// TwinCAT 3 PLC project FsControllerToolbox
// Title: FsControllerToolbox
// Company: FisoThemes
// Author: Goodwill Mzumala
// ProjectVersion: 0.4.0
// Description: A library of composable building blocks for modelling and building control systems in TwinCAT.
// ProgramVersion: 3.1.4024.0
// libraries:
//   FsCommon, * (FisoThemes)
//   Tc2_Math, * (Beckhoff Automation GmbH)
//   Tc2_Standard, * (Beckhoff Automation GmbH)
//   Tc2_System, * (Beckhoff Automation GmbH)
//   Tc3_Module, * (Beckhoff Automation GmbH)
// project tree:
//   Conditioning/DUTs/ E_DeadbandMode.TcTLEO
//   Conditioning/ FB_Clamp.TcPOU, FB_Deadband.TcPOU, FB_Hysteresis.TcPOU, FB_RateLimiter.TcPOU
//   Control/DUTs/ E_AntiWindupMode.TcTLEO, E_ControllerMode.TcTLEO
//   Control/ FB_ClampingIntegrator.TcPOU, FB_Differentiator.TcPOU, FB_ExtendedStateObserver.TcPOU (not stored), FB_Integrator.TcPOU, FB_LADRC.TcPOU (not stored), FB_LinearStateErrorFeedback.TcPOU, FB_PID.TcPOU (not stored), FB_ProportionalGain.TcPOU, FB_TrackingIntegrator.TcPOU
//   Filter/ FB_FirstOrderIIRFilter.TcPOU
//   / PlcTask.TcTTO
//   Internal/ PLAYGROUND.TcPOU (not stored)
//   Project Information/ F_GetCompany.TcPOU, F_GetTitle.TcPOU, F_GetVersion.TcPOU
//   Shared/ FB_SiComponent.TcPOU, FB_SisoComponent.TcPOU, FB_SoComponent.TcPOU
//   Shared/ITFs/ I_Bounded.TcIO, I_Component.TcIO, I_Resettable.TcIO, I_SiComponent.TcIO, I_SisoComponent.TcIO, I_SoComponent.TcIO
//   Signals/DUTs/ E_RampDirection.TcTLEO
//   Signals/ FB_GaussianNoise.TcPOU, FB_PeriodicSignal.TcPOU, FB_PWM.TcPOU, FB_Ramp.TcPOU, FB_RampProfile.TcPOU, FB_SawtoothWave.TcPOU, FB_SineWave.TcPOU, FB_SquareWave.TcPOU, FB_TriangleWave.TcPOU, FB_WhiteNoise.TcPOU
//   Signals/ITFs/ I_PeriodicSignal.TcIO
//   Simulation/ FB_FirstOrderPlant.TcPOU, FB_PadeDelay.TcPOU, FB_SecondOrderPlant.TcPOU
//   Transform/ FB_Bias.TcPOU, FB_Gain.TcPOU, FB_LinearScaler.TcPOU, FB_Quantizer.TcPOU
//   Version/ Global_Version.TcGVL
// real-time tasks:
//   TASK PlcTask: cycle T#10ms, priority 20, ADS port 350
//   TASK PlcTestTask: cycle T#10ms, priority 21, ADS port 351

CONFIGURATION FsControllerToolbox
    RESOURCE PLC ON TwinCAT3
        TASK PlcTask(INTERVAL := T#10ms, PRIORITY := 20);
        PROGRAM PLAYGROUND WITH PlcTask : PLAYGROUND;
    END_RESOURCE
END_CONFIGURATION

// ---- Conditioning/DUTs/E_DeadbandMode.TcTLEO
(*
Specifies the behaviour of :itf:`FB_Deadband` when the input is within the band.
*)
{attribute 'qualified_only'}
{attribute 'strict'}
{attribute 'to_string'}
TYPE E_DeadbandMode :
(
	Hold := 0, // Output holds its last value while the input is within the band.
	Zero := 1  // Output is set to zero while the input is within the band.
)BYTE;
END_TYPE

// ---- Control/DUTs/E_AntiWindupMode.TcTLEO
(*
Specifies the anti-windup behaviour of :class:`FB_ClampingIntegrator` when
saturation is detected via :attr:`~FB_ClampingIntegrator.ComparitorInput`.
*)
{attribute 'qualified_only'}
{attribute 'strict'}
{attribute 'to_string'}
TYPE E_AntiWindupMode :
(
	// Holds the integrator output at its current value while saturation is active.
	Hold := 0,
	// Zeroes the integrator output on the rising edge of saturation detection.
	Off  := 1
)BYTE;
END_TYPE

// ---- Control/DUTs/E_ControllerMode.TcTLEO
(* Specifies the operating mode of a controller. *)
{attribute 'qualified_only'}
{attribute 'strict'}
{attribute 'to_string'}
TYPE E_ControllerMode :
(
	// Output is computed from Setpoint and Feedback using the controller's algorithm.
	Auto 	:= 0,
	// Output tracks Setpoint directly.
	Manual	:= 1
)BYTE;
END_TYPE

// ---- Signals/DUTs/E_RampDirection.TcTLEO
(* Specifies the direction of a ramping signal. *)
{attribute 'qualified_only'}
{attribute 'strict'}
{attribute 'to_string'}
TYPE E_RampDirection :
(
	Rising   := 0, // Output increases over time.
	Falling  := 1  // Output decreases over time.
)BYTE;
END_TYPE

// ---- Version/Global_Version.TcGVL
{attribute 'TcGenerated'}
{attribute 'no-analysis'}
{attribute 'linkalways'}
// This function has been automatically generated from the project information.
VAR_GLOBAL CONSTANT
	{attribute 'const_non_replaced'}
	stLibVersion_FsControllerToolbox : ST_LibVersion := (iMajor := 0, iMinor := 4, iBuild := 0, iRevision := 0, nFlags := 0, sVersion := '0.4.0');
END_VAR

// ---- Shared/ITFs/I_Bounded.TcIO
(*
Exposes configurable upper and lower bounds for blocks with clamped output.

Implemented by blocks such as :class:`FB_ClampingIntegrator` and :class:`FB_Clamp`
to allow external configuration of their output limits.
*)
INTERFACE I_Bounded EXTENDS I_Component

(*
Gets or sets the upper bound.

This value could be clamped to be greater than or equal to :attr:`Minimum`.
Thus it is best practice to set this before :attr:`Minimum` to ensure the 
guard applies correctly.
*)
PROPERTY Maximum : LREAL
GET
END_GET
SET
END_SET
END_PROPERTY

(*
Gets or sets the lower bound.

This value could be clamped to be less than or equal to :attr:`Maximum`.
Thus it is best practice to set :attr:`Maximum` before this property to 
ensure the guard applies correctly.
*)
PROPERTY Minimum : LREAL
GET
END_GET
SET
END_SET
END_PROPERTY

END_INTERFACE

// ---- Shared/ITFs/I_Component.TcIO
(*
Base interface for all FsControllerToolbox components.

Extends ``__SYSTEM.IQueryInterface`` to allow runtime type checking via
``__QUERYINTERFACE``.
*)
INTERFACE I_Component EXTENDS __SYSTEM.IQueryInterface

END_INTERFACE

// ---- Shared/ITFs/I_Resettable.TcIO
(*
Interface for components that can be returned to a known initial state.

Implementors must define :meth:`Reset` to clear any internal state, such as
accumulators, filter history, or elapsed time, and restore the output to its
initial condition.
*)
INTERFACE I_Resettable EXTENDS __SYSTEM.IQueryInterface

(* Clears internal state and restores the component to its initial condition. *)
METHOD Reset
VAR_INPUT
END_VAR
END_METHOD

END_INTERFACE

// ---- Shared/ITFs/I_SiComponent.TcIO
(*
Interface for single-input controller toolbox components.

Implementors expose a write-only :attr:`Input` property. For components that
also produce an output signal, use :itf:`I_SisoComponent` instead.
*)
INTERFACE I_SiComponent

// Gets or sets the input to the component.
PROPERTY Input : LREAL
GET
END_GET
SET
END_SET
END_PROPERTY

END_INTERFACE

// ---- Shared/ITFs/I_SisoComponent.TcIO
(*
Interface for single-input single-output controller toolbox components.

Implementors expose a writable :attr:`Input` and a read-only :attr:`Output`,
both as ``LREAL``.
*)
INTERFACE I_SisoComponent EXTENDS I_Component

// Gets or sets the input to the component.
PROPERTY Input : LREAL
GET
END_GET
SET
END_SET
END_PROPERTY

// Gets the output produced by the component.
PROPERTY Output : LREAL
GET
END_GET
END_PROPERTY

END_INTERFACE

// ---- Shared/ITFs/I_SoComponent.TcIO
(*
Interface for single-output controller toolbox components.

Implementors expose a read-only :attr:`Output` property. For components that
also accept an input signal, use :itf:`I_SisoComponent` instead.
*)
INTERFACE I_SoComponent EXTENDS I_Component

// Gets the output produced by the component.
PROPERTY Output : LREAL
GET
END_GET
END_PROPERTY

END_INTERFACE

// ---- Signals/ITFs/I_PeriodicSignal.TcIO
(*
Base interface for periodic signal generators.

Implementors produce a cyclic output defined by :attr:`Period`, :attr:`Amplitude`,
:attr:`Bias`, and :attr:`Phase`.
*)
INTERFACE I_PeriodicSignal EXTENDS I_SoComponent

(*
Gets or sets the amplitude. 

The output swings between ``Bias + Amplitude`` and ``Bias - Amplitude``.
*)
PROPERTY Amplitude : LREAL
GET
END_GET
SET
END_SET
END_PROPERTY

(*
Gets or sets the bias.

This is a fixed offset added to the output, shifting the wave up or down.
*)
PROPERTY Bias : LREAL
GET
END_GET
SET
END_SET
END_PROPERTY

(* 
Gets or sets the period. 

This is the time taken to complete one full cycle.
*)
PROPERTY Period : LTIME
GET
END_GET
SET
END_SET
END_PROPERTY

(*
Gets or sets the phase offset in radians.

This shifts the wave horizontally. Negative values shift in the opposite direction.
*)
PROPERTY Phase : LREAL
GET
END_GET
SET
END_SET
END_PROPERTY

END_INTERFACE

// ---- Conditioning/FB_Clamp.TcPOU
(*
Clamps the input signal to the range [:attr:`Minimum`, :attr:`Maximum`].

Any input below :attr:`Minimum` is set to :attr:`Minimum`. Any input above
:attr:`Maximum` is set to :attr:`Maximum`. Inputs within the range pass
through unchanged.

.. note::
   The block is ``FINAL`` and must be instantiated, not extended.
   Use ``FB_init`` to set :attr:`fMaximum` and :attr:`fMinimum` at declaration time.
*)
{attribute 'enable_dynamic_creation'}
{attribute 'no_explicit_call' := 'direct call for this function block is not allowed'}
FUNCTION_BLOCK FINAL FB_Clamp EXTENDS FB_SisoComponent
IMPLEMENTS FsCommon.I_Runnable, I_Bounded
VAR
	_fMaximum  : LREAL; // Upper clamp bound. Clamped to >= Minimum.
	_fMinimum  : LREAL; // Lower clamp bound. Clamped to <= Maximum.
	_fResidual : LREAL; // Difference between the unclamped input and the clamped output.
END_VAR

METHOD FB_init : BOOL
VAR_INPUT
	bInitRetains : BOOL; // if TRUE, the retain variables are initialized (warm start / cold start)
	bInCopyCode  : BOOL;  // if TRUE, the instance afterwards gets moved into the copy code (online change)
	fMaximum     : LREAL; // Upper clamp bound.
	fMinimum     : LREAL; // Lower clamp bound.
END_VAR
THIS^.Maximum := fMaximum;
THIS^.Minimum := fMinimum;
END_METHOD

(*
Gets or sets the upper clamp bound.

Internally clamped to be greater than or equal to :attr:`Minimum`.
Set this before :attr:`Minimum` to ensure the guard applies correctly.
*)
PROPERTY Maximum : LREAL
GET
Maximum := THIS^._fMaximum;
END_GET
SET
THIS^._fMaximum := MAX(THIS^._fMinimum, Maximum);
END_SET
END_PROPERTY

(*
Gets or sets the lower clamp bound.

Internally clamped to be less than or equal to :attr:`Maximum`.
Set :attr:`Maximum` before this property to ensure the guard applies correctly.
*)
PROPERTY Minimum : LREAL
GET
Minimum := THIS^._fMinimum;
END_GET
SET
THIS^._fMinimum := MIN(THIS^._fMaximum, Minimum);
END_SET
END_PROPERTY

(* Gets the difference between the unclamped input and the clamped output. Zero when the input is within [:attr:`Minimum`, :attr:`Maximum`]. *)
PROPERTY Residual : LREAL
GET
Residual := THIS^._fResidual;
END_GET
END_PROPERTY

(* Clamps the current input to [:attr:`Minimum`, :attr:`Maximum`]. *)
METHOD Run
VAR_INPUT
END_VAR
THIS^._fOutput 	 := LIMIT(THIS^._fMinimum, THIS^._fInput, THIS^._fMaximum);
THIS^._fResidual := THIS^._fInput - THIS^._fOutput;
END_METHOD

END_FUNCTION_BLOCK

// ---- Shared/FB_SisoComponent.TcPOU
(*
Abstract function block providing :attr:`Input` and :attr:`Output` properties
for single-input single-output controller toolbox components.

.. NOTE::
   Direct calls to this function block are not permitted (``no_explicit_call``).
*)
{attribute 'no_explicit_call' := 'direct call for this function block is not allowed'}
FUNCTION_BLOCK ABSTRACT FB_SisoComponent
IMPLEMENTS I_SisoComponent, I_SiComponent, I_SoComponent
VAR
	_fInput 	: LREAL;
	_fOutput 	: LREAL;
END_VAR

(* Gets or sets the input to the component.*)
PROPERTY Input : LREAL
GET
Input := THIS^._fInput;
END_GET
SET
THIS^._fInput := Input;
END_SET
END_PROPERTY

(* Gets the output produced by the component.*)
PROPERTY Output : LREAL
GET
Output := THIS^._fOutput;
END_GET
END_PROPERTY

END_FUNCTION_BLOCK

// ---- Conditioning/FB_Deadband.TcPOU
(*
Suppresses small input signals within a configurable band.

When the input falls within [:attr:`Minimum`, :attr:`Maximum`], the output
is either zeroed or held at its last value depending on :attr:`Mode`. Outside
the band the input passes through unchanged.

.. note::
   The block is ``FINAL`` and must be instantiated, not extended.
   Use ``FB_init`` to set :attr:`fMinimum`, :attr:`fMaximum`, and :attr:`eMode`
   at declaration time.
*)
{attribute 'enable_dynamic_creation'}
{attribute 'no_explicit_call' := 'direct call for this function block is not allowed'}
FUNCTION_BLOCK FINAL FB_Deadband EXTENDS FB_SisoComponent
IMPLEMENTS FsCommon.I_Runnable, I_Resettable
VAR
	_fMinimum  : LREAL; // Lower bound of the deadband. Clamped to <= Maximum.
	_fMaximum  : LREAL; // Upper bound of the deadband. Clamped to >= Minimum.
	_eMode     : E_DeadbandMode; // Output behaviour when input is within the band.
	_bIsActive : BOOL; // TRUE when input is within deadband [Minimum..:=Maximum].
END_VAR

METHOD FB_init : BOOL
VAR_INPUT
	bInitRetains : BOOL;  // if TRUE, the retain variables are initialized (warm start / cold start)
	bInCopyCode  : BOOL;  // if TRUE, the instance afterwards gets moved into the copy code (online change)
	fMaximum     : LREAL; // Upper bound of the deadband.
	fMinimum     : LREAL; // Lower bound of the deadband.
	eMode        : E_DeadbandMode; // Output behaviour when the input is within the band.
END_VAR
THIS^.Maximum  := fMaximum;
THIS^.Minimum  := fMinimum;
THIS^._eMode   := eMode;
END_METHOD

(*
Gets whether the input is within the deadband's bounds.

``TRUE`` when the output is being held or zeroed.
*)
PROPERTY IsActive : BOOL
GET
IsActive := THIS^._bIsActive;
END_GET
END_PROPERTY

(*
Gets or sets the upper bound of the deadband.

Internally clamped to be greater than or equal to :attr:`Minimum`.
Set this before :attr:`Minimum` to ensure the guard applies correctly.
*)
PROPERTY Maximum : LREAL
GET
Maximum := THIS^._fMaximum;
END_GET
SET
THIS^._fMaximum := MAX(THIS^._fMinimum, Maximum);
END_SET
END_PROPERTY

(*
Gets or sets the lower bound of the deadband.

Internally clamped to be less than or equal to :attr:`Maximum`.
Set :attr:`Maximum` before this property to ensure the guard applies correctly.
*)
PROPERTY Minimum : LREAL
GET
Minimum := THIS^._fMinimum;
END_GET
SET
THIS^._fMinimum := MIN(THIS^._fMaximum, Minimum);
END_SET
END_PROPERTY

(*
Gets or sets the output behaviour when the input is within the band.

:attr:`~E_DeadbandMode.Zero` sets the output to zero. 
:attr:`~E_DeadbandMode.Hold` retains the last output value. 

Changes take effect on th next :meth:`Run` call.
*)
PROPERTY Mode : E_DeadbandMode
GET
Mode := THIS^._eMode;
END_GET
SET
THIS^._eMode := Mode;
END_SET
END_PROPERTY

(* 
Resets the output to a value consistent with the current mode. 

In :attr:`~E_DeadbandMode.Zero` mode the output is set to zero.
In :attr:`~E_DeadbandMode.Hold` mode the output is set to the current input.
*)
METHOD Reset
VAR_INPUT
END_VAR
CASE THIS^._eMode OF
	E_DeadbandMode.Hold:
		THIS^._fOutput := THIS^._fInput;
	E_DeadbandMode.Zero:
		THIS^._fOutput := 0;
END_CASE
END_METHOD

(* Applies the deadband to the current input. *)
METHOD Run
VAR_INPUT
END_VAR
THIS^._fMaximum := MAX(THIS^._fMinimum, THIS^._fMaximum);
THIS^._fMinimum := MIN(THIS^._fMinimum, THIS^._fMaximum);

THIS^._bIsActive := THIS^._fInput >= THIS^._fMinimum AND THIS^._fInput <= THIS^._fMaximum;

IF THIS^._bIsActive  THEN
    CASE THIS^._eMode OF
        E_DeadbandMode.Zero:
            THIS^._fOutput := 0;
        E_DeadbandMode.Hold:
            ; // Output retains its last value.
    END_CASE
ELSE
    THIS^._fOutput := THIS^._fInput;
END_IF
END_METHOD

END_FUNCTION_BLOCK

// ---- Conditioning/FB_Hysteresis.TcPOU
(*
Implements a hysteresis controller with two thresholds and latching behaviour.

The output switches low when the input rises above :attr:`UpperThreshold` and
switches high when the input falls below :attr:`LowerThreshold`. Between the
two thresholds the output latches at its current state.

This convention suits heating applications, the output drives a heater that
turns on when the process falls below the lower threshold and off when it
exceeds the upper threshold.

.. note::
   The block is ``FINAL`` and must be instantiated, not extended.
   Use ``FB_init`` to set :attr:`fUpperThreshold` and :attr:`fLowerThreshold`
   at declaration time.
*)
{attribute 'no_assign'}
{attribute 'enable_dynamic_creation'}
{attribute 'no_explicit_call' := 'direct call for this function block is not allowed'}
FUNCTION_BLOCK FINAL FB_Hysteresis EXTENDS FB_SiComponent
IMPLEMENTS FsCommon.I_Runnable, I_Resettable
VAR
	_fUpperThreshold : LREAL; // Input level above which the output switches low.
	_fLowerThreshold : LREAL; // Input level below which the output switches high.
	_bOutput         : BOOL;  // Current output state.
END_VAR

METHOD FB_init : BOOL
VAR_INPUT
	bInitRetains 	 : BOOL; // if TRUE, the retain variables are initialized (warm start / cold start)
	bInCopyCode 	 : BOOL;  // if TRUE, the instance afterwards gets moved into the copy code (online change)
	fUpperThreshold  : LREAL; // Input level above which the output switches low.
	fLowerThreshold  : LREAL; // Input level below which the output switches high.
END_VAR
THIS^._fUpperThreshold := fUpperThreshold;
THIS^._fLowerThreshold := fLowerThreshold;
END_METHOD

(*
Gets or sets the lower threshold.

When the input falls below this value the output switches high. Must be less
than :attr:`UpperThreshold` for correct operation.
*)
PROPERTY LowerThreshold : LREAL
GET
LowerThreshold := THIS^._fLowerThreshold;
END_GET
SET
THIS^._fLowerThreshold := LowerThreshold;
END_SET
END_PROPERTY

(*
Gets the current output state. 

TRUE when the process is below :attr:`LowerThreshold`.
FALSE when above :attr:`UpperThreshold`.
*)
PROPERTY Output : BOOL
GET
Output := THIS^._bOutput;
END_GET
END_PROPERTY

(*
Evaluates the current input against the thresholds and sets the output immediately,
rather than waiting for the input to cross a threshold.

If the input is above :attr:`UpperThreshold` the output is set low. If below
:attr:`LowerThreshold` the output is set high. If between the two thresholds
the output defaults to low as a safe state.
*)
METHOD Reset
VAR_INPUT
END_VAR
THIS^._bOutput := THIS^._fInput < THIS^._fLowerThreshold;
END_METHOD

(* Evaluates the input against the thresholds and updates the output. *)
METHOD Run
VAR_INPUT
END_VAR
IF THIS^._fInput > THIS^._fUpperThreshold THEN
	THIS^._bOutput := FALSE;
ELSIF THIS^._fInput < THIS^._fLowerThreshold THEN
	THIS^._bOutput := TRUE;
END_IF
END_METHOD

(*
Gets or sets the upper threshold.

When the input rises above this value the output switches low. Must be greater
than :attr:`LowerThreshold` for correct operation.
*)
PROPERTY UpperThreshold : LREAL
GET
UpperThreshold := THIS^._fUpperThreshold;
END_GET
SET
THIS^._fUpperThreshold := UpperThreshold;
END_SET
END_PROPERTY

END_FUNCTION_BLOCK

// ---- Shared/FB_SiComponent.TcPOU
(*
Abstract function block providing an :attr:`Input` property for single-input
controller toolbox components.

Concrete implementations read from ``_fInput`` to consume the signal written
by the caller.

.. note::
   Direct calls to this function block are not permitted (``no_explicit_call``).
   Extend it and call the derived block instead.
*)
{attribute 'no_explicit_call' := 'direct call for this function block is not allowed'}
FUNCTION_BLOCK ABSTRACT FB_SiComponent
IMPLEMENTS I_SiComponent
VAR
    _fInput : LREAL;
END_VAR

(* Gets or sets the input to the component.*)
PROPERTY Input : LREAL
GET
Input := THIS^._fInput;
END_GET
SET
THIS^._fInput := Input;
END_SET
END_PROPERTY

END_FUNCTION_BLOCK

// ---- Conditioning/FB_RateLimiter.TcPOU
(*
Limits the rate of change of the input signal.

The output tracks the input but cannot change faster than :attr:`RisingLimit`
units per second when increasing, or :attr:`FallingLimit` units per second when
decreasing. A limit of zero removes the restriction in that direction, allowing
the output to change freely.

Calling :meth:`Reset` snaps the output to the current input immediately.

.. note::
   The block is ``FINAL`` and must be instantiated, not extended.
   Use ``FB_init`` to set :attr:`fRisingLimit` and :attr:`fFallingLimit` at
   declaration time.
*)
{attribute 'enable_dynamic_creation'}
{attribute 'no_explicit_call' := 'direct call for this function block is not allowed'}
FUNCTION_BLOCK FINAL FB_RateLimiter EXTENDS FB_SisoComponent
IMPLEMENTS FsCommon.I_Runnable, I_Resettable
VAR
	_fRisingLimit  : LREAL; // Maximum rate of increase in units per second. Zero means no limit.
	_fFallingLimit : LREAL; // Maximum rate of decrease in units per second. Zero means no limit.
END_VAR

(*
Gets or sets the maximum rate of decrease in units per second.

The output will not fall faster than this value regardless of how quickly
the input changes. A value of zero removes the falling limit entirely.
Values below zero are clamped to zero.
*)
PROPERTY FallingLimit : LREAL
GET
FallingLimit := THIS^._fFallingLimit;
END_GET
SET
THIS^._fFallingLimit := MAX(0, FallingLimit);
END_SET
END_PROPERTY

METHOD FB_init : BOOL
VAR_INPUT
	bInitRetains   : BOOL; // if TRUE, the retain variables are initialized (warm start / cold start)
	bInCopyCode    : BOOL;  // if TRUE, the instance afterwards gets moved into the copy code (online change)
	fRisingLimit   : LREAL; // Maximum rate of increase in units per second. Zero means no limit.
	fFallingLimit  : LREAL; // Maximum rate of decrease in units per second. Zero means no limit.
END_VAR
THIS^.RisingLimit  := fRisingLimit;
THIS^.FallingLimit := fFallingLimit;
END_METHOD

(* Snaps the output to the current input, bypassing the rate limit. *)
METHOD Reset
VAR_INPUT
END_VAR
THIS^._fOutput := THIS^._fInput;
END_METHOD

(*
Gets or sets the maximum rate of increase in units per second.

The output will not rise faster than this value regardless of how quickly
the input changes. A value of zero removes the rising limit entirely.
Values below zero are clamped to zero.
*)
PROPERTY RisingLimit : LREAL
GET
RisingLimit := THIS^._fRisingLimit;
END_GET
SET
THIS^._fRisingLimit := MAX(0, RisingLimit);
END_SET
END_PROPERTY

(*
Advances the rate limiter by one time step.

.. note::
   Must be called once per cycle on a single PLC task. If the measured cycle
   time is zero the method returns early without updating the output.
*)
METHOD Run
VAR_INST
	{attribute 'hide'}
	bInit       : BOOL := TRUE;
	{attribute 'hide'}
	fT          : LREAL;
	{attribute 'hide'}
	fbTaskCycle : FsCommon.FB_PlcTaskCycleChangeDetector(0);
END_VAR
VAR
	fDelta    	: LREAL;
	fMaxDelta 	: LREAL;
END_VAR
IF bInit THEN
	fT := TO_LREAL(FsCommon.F_GetCurrentTaskCycleTime()) / TO_LREAL(LTIME#1S);
	RETURN(bInit := fT <= 0);
	fbTaskCycle.TaskIndex := FsCommon.F_GetCurrentTaskIndex();
	THIS^._fOutput := THIS^._fInput;
	RETURN;
END_IF

RETURN(NOT fbTaskCycle.HasChanged);

THIS^._fRisingLimit  := MAX(0, THIS^._fRisingLimit);
THIS^._fFallingLimit := MAX(0, THIS^._fFallingLimit);

fDelta := THIS^._fInput - THIS^._fOutput;

IF fDelta > 0 AND THIS^._fRisingLimit > 0 THEN
	fMaxDelta      := THIS^._fRisingLimit * fT;
	THIS^._fOutput := THIS^._fOutput + MIN(fDelta, fMaxDelta);
ELSIF fDelta < 0 AND THIS^._fFallingLimit > 0 THEN
	fMaxDelta      := THIS^._fFallingLimit * fT;
	THIS^._fOutput := THIS^._fOutput - MIN(ABS(fDelta), fMaxDelta);
ELSE
	THIS^._fOutput := THIS^._fInput;
END_IF
END_METHOD

END_FUNCTION_BLOCK

// ---- Control/FB_ClampingIntegrator.TcPOU
(*
Integrates the input error signal with comparator-based anti-windup.

Extends :class:`FB_Integrator` by suppressing integration when the
:attr:`ComparatorInput` indicates saturation and the input would push
further into saturation. The suppression behaviour is controlled by :attr:`Mode`.

:attr:`ComparatorInput` is typically the :attr:`~FB_Clamp.Residual` of an
:class:`FB_Clamp` block placed after the PID summation.

.. note::
   Set :attr:`Maximum` before :attr:`Minimum` to ensure the clamp guard applies
   correctly.

   Use ``FB_init`` to set :attr:`tTn` and :attr:`eMode` at declaration time.
*)
{attribute 'no_assign'}
{attribute 'enable_dynamic_creation'}
{attribute 'no_explicit_call' := 'direct call for this function block is not allowed'}
FUNCTION_BLOCK FINAL FB_ClampingIntegrator EXTENDS FB_Integrator
VAR
	_fComparatorInput  : LREAL;
	_bAntiWindupActive : BOOL; // TRUE when the output is saturated and integration is halted.
	_eMode			   : E_AntiWindupMode; // The integrator behaviour during saturation.
END_VAR

(* Gets whether the output is currently saturated and integration is halted. *)
PROPERTY AntiWindupActive : BOOL
GET
AntiWindupActive := THIS^._bAntiWindupActive;
END_GET
END_PROPERTY

(*
Gets or sets the comparator input.

This is typically the :attr:`~FB_Clamp.Residual` of an :class:`FB_Clamp` block
placed after the PID summation. A positive value indicates the unsaturated sum
exceeded the clamp maximum; a negative value indicates it fell below the clamp
minimum. When this value and :attr:`Input` have the same sign, integration is
suppressed according to :attr:`Mode`.
*)
PROPERTY ComparatorInput : LREAL
GET
ComparatorInput := THIS^._fComparatorInput;
END_GET
SET
THIS^._fComparatorInput := ComparatorInput;
END_SET
END_PROPERTY

METHOD FB_init : BOOL
VAR_INPUT
	bInitRetains : BOOL;  // if TRUE, the retain variables are initialized (warm start / cold start)
	bInCopyCode  : BOOL;  // if TRUE, the instance afterwards gets moved into the copy code (online change)
	tTn          : LTIME; // Integral action time. LTIME#0 disables integration.
	eMode		 : E_AntiWindupMode; // The integrator behaviour during saturation.
END_VAR
THIS^._eMode := eMode;
END_METHOD

(*
Gets or sets the anti-windup mode.

Controls the integrator behaviour when saturation is detected via
:attr:`ComparatorInput`. See :class:`E_AntiWindupMode` for available modes.
*)
PROPERTY Mode : E_AntiWindupMode
GET
Mode := THIS^._eMode;
END_GET
SET
THIS^._eMode := Mode;
END_SET
END_PROPERTY

(* Clears the integrator state, output, and anti-windup flag. *)
METHOD Reset
VAR_INPUT
END_VAR
THIS^._fOutput           := 0;
THIS^._bAntiWindupActive := FALSE;
END_METHOD

(*
Advances the clamping integrator by one time step.

.. note::
   Must be called once per cycle on a single PLC task. If :attr:`Tn` is
   ``LTIME#0`` the output is set to zero and anti-windup is cleared.
*)
METHOD Run
VAR_INST
	{attribute 'hide'}
	bInit       : BOOL := TRUE;
	{attribute 'hide'}
	fT          : LREAL;
	{attribute 'hide'}
	fbTaskCycle : FsCommon.FB_PlcTaskCycleChangeDetector(0);
	{attribute 'hide'}
	fbTrig 		: F_TRIG;
END_VAR
VAR
END_VAR
IF bInit THEN
	fT := TO_LREAL(FsCommon.F_GetCurrentTaskCycleTime()) / TO_LREAL(LTIME#1S);
	RETURN(bInit := fT <= 0);
	fbTaskCycle.TaskIndex := FsCommon.F_GetCurrentTaskIndex();
END_IF

RETURN(NOT fbTaskCycle.HasChanged);

THIS^._fMaximum := MAX(THIS^._fMinimum, THIS^._fMaximum);
THIS^._fMinimum := MIN(THIS^._fMinimum, THIS^._fMaximum);

IF FsCommon.F_ResetOnTrue(THIS^._bSync) THEN
	THIS^._fOutput := LIMIT(THIS^._fMinimum, THIS^._fSync, THIS^._fMaximum);
END_IF

IF THIS^._tTn = LTIME#0S THEN
	THIS^._fOutput           := 0;
	THIS^._bAntiWindupActive := FALSE;
	RETURN;
END_IF

THIS^._bAntiWindupActive := (THIS^._fComparatorInput > 0.0 AND THIS^._fInput > 0.0)
							 OR 
                            (THIS^._fComparatorInput < 0.0 AND THIS^._fInput < 0.0);
							
fbTrig(CLK := THIS^._bAntiWindupActive);
IF fbTrig.Q AND THIS^._eMode = E_AntiWindupMode.Off THEN 
	THIS^._bAntiWindupActive := TRUE;
END_IF
							
IF THIS^._bAntiWindupActive THEN
	CASE THIS^._eMode OF 
		E_AntiWindupMode.Hold:;
		E_AntiWindupMode.Off:
			THIS^._fOutput := 0.0;
	END_CASE
ELSE
	THIS^._fOutput := LIMIT(
		THIS^._fMinimum, 
		THIS^._fOutput + (1.0 / (TO_LREAL(THIS^._tTn) / TO_LREAL(LTIME#1S))) * THIS^._fInput * fT,
		THIS^._fMaximum
	);
END_IF
END_METHOD

END_FUNCTION_BLOCK

// ---- Control/FB_Integrator.TcPOU
(*
Integrates the input error signal over time.

The output accumulates the input scaled by the integral gain :math:`K_i = 1 / T_n`,
and is clamped to [:attr:`Minimum`, :attr:`Maximum`] on every cycle.
Setting :attr:`Tn` to ``LTIME#0`` disables integration, setting the output to zero.

Use :meth:`Sync` to preset the integrator state for bumpless transfer when
switching from manual to automatic mode.

.. note::
   Set :attr:`Maximum` before :attr:`Minimum` to ensure the clamp guard applies
   correctly.

   Use ``FB_init`` to set :attr:`tTn` at declaration time.
*)
{attribute 'no_assign'}
{attribute 'enable_dynamic_creation'}
{attribute 'no_explicit_call' := 'direct call for this function block is not allowed'}
FUNCTION_BLOCK FB_Integrator EXTENDS FB_SisoComponent
IMPLEMENTS FsCommon.I_Runnable, I_Resettable, I_Bounded
VAR
	_tTn   		: LTIME; // Integral action time (Tn).
	_bSync 		: BOOL;  // Triggers a bumpless transfer on the next Run call.
	_fSync 		: LREAL; // Target integrator state for bumpless transfer.
	_fMaximum   : LREAL := FsCommon.GVL_TypeValueLimits.LREAL_MAX; // Upper output clamp. Clamped to >= Minimum.
	_fMinimum   : LREAL := FsCommon.GVL_TypeValueLimits.LREAL_MIN; // Lower output clamp. Clamped to <= Maximum.
END_VAR

METHOD FB_init : BOOL
VAR_INPUT
	bInitRetains : BOOL;  // if TRUE, the retain variables are initialized (warm start / cold start)
	bInCopyCode  : BOOL;  // if TRUE, the instance afterwards gets moved into the copy code (online change)
	tTn          : LTIME; // Integral action time. LTIME#0 disables integration.
END_VAR
THIS^._tTn := tTn;
END_METHOD

(*
Gets or sets the upper output clamp.

Internally clamped to be greater than or equal to :attr:`Minimum`.
Set this before :attr:`Minimum` to ensure the guard applies correctly.
*)
PROPERTY Maximum : LREAL
GET
Maximum := THIS^._fMaximum;
END_GET
SET
THIS^._fMaximum := MAX(THIS^._fMinimum, Maximum);
END_SET
END_PROPERTY

(*
Gets or sets the lower output clamp.

Internally clamped to be less than or equal to :attr:`Maximum`.
Set :attr:`Maximum` before this property to ensure the guard applies correctly.
*)
PROPERTY Minimum : LREAL
GET
Minimum := THIS^._fMinimum;
END_GET
SET
THIS^._fMinimum := MIN(THIS^._fMaximum, Minimum);
END_SET
END_PROPERTY

(* Clears the integrator state and output. *)
METHOD Reset
VAR_INPUT
END_VAR
THIS^._fOutput := 0;
END_METHOD

(*
Advances the integrator by one time step.

.. note::
   Must be called once per cycle on a single PLC task. If :attr:`Tn` is
   ``LTIME#0`` the output is set to zero.
*)
METHOD Run
VAR_INST
	{attribute 'hide'}
	bInit       : BOOL := TRUE;
	{attribute 'hide'}
	fT          : LREAL;
	{attribute 'hide'}
	fbTaskCycle : FsCommon.FB_PlcTaskCycleChangeDetector(0);
END_VAR
IF bInit THEN
	fT := TO_LREAL(FsCommon.F_GetCurrentTaskCycleTime()) / TO_LREAL(LTIME#1S);
	RETURN(bInit := fT <= 0);
	fbTaskCycle.TaskIndex := FsCommon.F_GetCurrentTaskIndex();
END_IF

RETURN(NOT fbTaskCycle.HasChanged);

THIS^._fMaximum := MAX(THIS^._fMinimum, THIS^._fMaximum);
THIS^._fMinimum := MIN(THIS^._fMinimum, THIS^._fMaximum);

IF FsCommon.F_ResetOnTrue(THIS^._bSync) THEN
	THIS^._fOutput := THIS^._fSync;
END_IF

IF THIS^._tTn = LTIME#0S THEN
	THIS^._fOutput := 0;
	RETURN;
END_IF

THIS^._fOutput := LIMIT(
	THIS^._fMinimum, 
	THIS^._fOutput + 
		(1.0 / (TO_LREAL(THIS^._tTn) / TO_LREAL(LTIME#1S))) * THIS^._fInput * fT,
	THIS^._fMaximum
);
END_METHOD

(*
Forces the integrator state to a given value on the next :meth:`Run` call.

Use this for bumpless transfer when switching from manual to automatic mode,
to prevent a sudden jump in output.
*)
METHOD Sync
VAR_INPUT
	// Target integrator state.
	fValue : LREAL; 
END_VAR
THIS^._bSync := TRUE;
THIS^._fSync := fValue;
END_METHOD

(*
Gets or sets the integral action time (Tn).

This controls how aggressively the integrator responds to sustained error.
A shorter value increases integral action. Setting it to ``LTIME#0`` disables
integration entirely, setting the output to zero.
*)
PROPERTY Tn : LTIME
GET
Tn := THIS^._tTn;
END_GET
SET
THIS^._tTn := Tn;
END_SET
END_PROPERTY

END_FUNCTION_BLOCK

// ---- Control/FB_Differentiator.TcPOU
(*
Differentiates the input signal with an optional first-order damping filter.

The transfer function is:

.. math::

   D(s) = \frac{T_v \cdot s}{T_d \cdot s + 1}

where :math:`T_v` is :attr:`Tv` and :math:`T_d` is :attr:`Td`. The filter is
discretised using the Tustin (bilinear) method.

Setting :attr:`Tv` to ``LTIME#0`` disables the derivative term entirely.
Setting :attr:`Td` to ``LTIME#0`` removes the damping filter, giving a pure
derivative. This is not recommended in practice due to noise sensitivity.

.. note::
   If derivative kick on setpoint steps is undesirable, pass the negated
   process variable as :attr:`Input` rather than the full error. The integrator
   should still receive the full error signal.

   The block is ``FINAL`` and must be instantiated, not extended.
   Use ``FB_init`` to set :attr:`tTv` and :attr:`tTd` at declaration time.
*)
{attribute 'no_assign'}
{attribute 'enable_dynamic_creation'}
{attribute 'no_explicit_call' := 'direct call for this function block is not allowed'}
FUNCTION_BLOCK FINAL FB_Differentiator EXTENDS FB_SisoComponent
IMPLEMENTS FsCommon.I_Runnable, I_Resettable
VAR
	_tTv          : LTIME; // Rate time (Tv). Determines derivative action strength.
	_tTd          : LTIME; // Damping time (Td). Filters the derivative signal to reduce noise sensitivity.
	_fPrevInput   : LREAL; // Input from the previous cycle.
	_fFilterState : LREAL; // Internal state of the damping filter.
END_VAR

METHOD FB_init : BOOL
VAR_INPUT
	bInitRetains : BOOL; // if TRUE, the retain variables are initialized (warm start / cold start)
	bInCopyCode  : BOOL;  // if TRUE, the instance afterwards gets moved into the copy code (online change)
	tTv          : LTIME; // Rate time. T#0S disables the derivative term entirely.
	tTd          : LTIME; // Damping time. LTIME#0 means no filtering (pure derivative).
END_VAR
THIS^._tTv := tTv;
THIS^._tTd := tTd;
END_METHOD

(*
Clears the filter state and output. 
Sets the previous input to the current input to avoid a spike on the next :meth:`Run` call. 
*)
METHOD Reset
VAR_INPUT
END_VAR
THIS^._fFilterState := 0;
THIS^._fPrevInput   := THIS^._fInput;
THIS^._fOutput      := 0;
END_METHOD

(*
Advances the differentiator by one time step.

On the first call the cycle time is measured, the filter state is initialised,
and the method returns early without producing an output. This prevents a spike
caused by an uninitialised previous input.

.. note::
   Must be called once per cycle on a single PLC task. If :attr:`Tv` is
   ``LTIME#0`` the output is held at zero.
*)
METHOD Run
VAR_INST
	{attribute 'hide'}
	bInit       : BOOL := TRUE;
	{attribute 'hide'}
	fT          : LREAL;
	{attribute 'hide'}
	fbTaskCycle : FsCommon.FB_PlcTaskCycleChangeDetector(0);
END_VAR
VAR
	fTv            : LREAL;
	fTd            : LREAL;
	fDen           : LREAL;
	fAlpha         : LREAL;
	fRawDerivative : LREAL;
END_VAR
IF bInit THEN
	fT := TO_LREAL(FsCommon.F_GetCurrentTaskCycleTime()) / TO_LREAL(LTIME#1S);
	RETURN(bInit := fT <= 0);
	fbTaskCycle.TaskIndex := FsCommon.F_GetCurrentTaskIndex();
	THIS^._fPrevInput     := THIS^._fInput;
	THIS^._fFilterState   := 0;
	RETURN;
END_IF

RETURN(NOT fbTaskCycle.HasChanged);

IF THIS^._tTv = LTIME#0S THEN
	THIS^._fOutput    := 0;
	THIS^._fPrevInput := THIS^._fInput;
	RETURN;
END_IF

fTv := TO_LREAL(THIS^._tTv) / TO_LREAL(LTIME#1S);
fTd := TO_LREAL(THIS^._tTd) / TO_LREAL(LTIME#1S);

fRawDerivative := fTv * (THIS^._fInput - THIS^._fPrevInput) / fT;

IF THIS^._tTd = LTIME#0S THEN
	THIS^._fOutput := fRawDerivative;
ELSE
	fDen                := fTd + fT / 2.0;
	fAlpha              := (fTd - fT / 2.0) / fDen;
	THIS^._fFilterState := fAlpha * THIS^._fFilterState + (1.0 - fAlpha) * fRawDerivative;
	THIS^._fOutput      := THIS^._fFilterState;
END_IF

THIS^._fPrevInput := THIS^._fInput;
END_METHOD

(*
Gets or sets the damping time (Td).

This filters the derivative signal to reduce sensitivity to noise. A longer
value gives more filtering but reduces derivative effectiveness. Setting it
to ``LTIME#0`` removes the filter entirely, giving a pure derivative (not
recommended in practice due to noise sensitivity).
*)
PROPERTY Td : LTIME
GET
Td := THIS^._tTd;
END_GET
SET
THIS^._tTd := Td;
END_SET
END_PROPERTY

(*
Gets or sets the rate time (Tv).

This controls how strongly the block reacts to changes in the input. A longer
value increases derivative action. Setting it to ``LTIME#0`` disables the
derivative term entirely, holding the output at zero.
*)
PROPERTY Tv : LTIME
GET
Tv := THIS^._tTv;
END_GET
SET
THIS^._tTv := Tv;
END_SET
END_PROPERTY

END_FUNCTION_BLOCK

// ---- Control/FB_LinearStateErrorFeedback.TcPOU
(*
Computes the control output for a Linear Active Disturbance Rejection Controller (LADRC).

The control law is:

.. math::

   u_0 = \omega_c \cdot (SP - z_1) + u_i

   u = \frac{u_0 - z_2}{b_0}

where :math:`u_0` is the error feedback, :math:`u_i` is the integral correction
from an external integrator, :math:`z_2` cancels the estimated disturbance from
:class:`FB_ExtendedStateObserver`, and dividing by :attr:`B0` scales the output
to the plant's input range.

If :attr:`B0` is zero the output is held at zero.

.. note::
   The block is ``FINAL`` and must be instantiated, not extended.
   Use ``FB_init`` to set :attr:`fWc` and :attr:`fB0` at declaration time.
*)
{attribute 'no_assign'}
{attribute 'enable_dynamic_creation'}
{attribute 'no_explicit_call' := 'direct call for this function block is not allowed'}
FUNCTION_BLOCK FINAL FB_LinearStateErrorFeedback EXTENDS FB_SoComponent
IMPLEMENTS FsCommon.I_Runnable, I_Resettable
VAR
	_fWc       : LREAL; // Controller bandwidth in rad/s.
	_fB0       : LREAL; // Estimated plant gain.
	_fSetpoint : LREAL; // Desired process output (SP).
	_fZ1       : LREAL; // Estimated process output from the observer.
	_fZ2       : LREAL; // Estimated total disturbance from the observer.
	_fIntegral : LREAL; // Integral correction from the external integrator.
END_VAR

(*
Gets or sets the estimated plant gain (b0).

Must be non-zero. A value of zero disables the control output entirely.
See :attr:`~FB_ADRC.B0` for guidance on how to estimate this value.
*)
PROPERTY B0 : LREAL
GET
B0 := THIS^._fB0;
END_GET
SET
THIS^._fB0 := B0;
END_SET
END_PROPERTY

METHOD FB_init : BOOL
VAR_INPUT
	bInitRetains : BOOL; // if TRUE, the retain variables are initialized (warm start / cold start)
	bInCopyCode : BOOL;  // if TRUE, the instance afterwards gets moved into the copy code (online change)
	fWc          : LREAL; // Controller bandwidth in rad/s.
	fB0          : LREAL; // Estimated plant gain.
END_VAR
THIS^._fWc := fWc;
THIS^._fB0 := fB0;
END_METHOD

(*
Gets or sets the integral correction.

Set this to the integrator output before calling :meth:`Run`. 
*)
PROPERTY Integral : LREAL
GET
Integral := THIS^._fIntegral;
END_GET
SET
THIS^._fIntegral := Integral;
END_SET
END_PROPERTY

(* Sets the output to zero. *)
METHOD Reset
VAR_INPUT
END_VAR
THIS^._fOutput := 0;
END_METHOD

(*
Computes the control output for the current cycle.

.. note::
   Must be called once per cycle on a single PLC task.
   If :attr:`b0` is zero the output is held at zero.
*)
METHOD Run
VAR
END_VAR
RETURN(THIS^._fb0 = 0);

THIS^._fOutput :=
    ((THIS^._fWc * (THIS^._fSetpoint - THIS^._fZ1)) + THIS^._fIntegral - THIS^._fZ2)
    / THIS^._fB0;
END_METHOD

(* Gets or sets the setpoint. This is the desired process output. *)
PROPERTY Setpoint : LREAL
GET
Setpoint := THIS^._fSetpoint;
END_GET
SET
THIS^._fSetpoint := Setpoint;
END_SET
END_PROPERTY

(*
Gets or sets the controller bandwidth in rad/s.

Controls how fast the closed loop responds to setpoint changes. A higher value
gives a faster response but risks overshoot and sensitivity to noise. Start with
a low value and increase until the response is satisfactory.

For a process that should settle in roughly 10 seconds, a starting value of
``Wc = 0.5`` rad/s is reasonable.
*)
PROPERTY Wc : LREAL
GET
Wc := THIS^._fWc;
END_GET
SET
THIS^._fWc := Wc;
END_SET
END_PROPERTY

(* 
Gets or sets the estimated process output from :class:`FB_ExtendedStateObserver`. 

Set this to ``Z1`` before calling :meth:`Run`.
*)
PROPERTY Z1 : LREAL
GET
Z1 := THIS^._fZ1;
END_GET
SET
THIS^._fZ1 := Z1;
END_SET
END_PROPERTY

(*
Gets or sets the estimated total disturbance from :class:`FB_ExtendedStateObserver`. 

Set this to ``Z2`` before calling :meth:`Run`.
*)
PROPERTY Z2 : LREAL
GET
Z2 := THIS^._fZ2;
END_GET
SET
THIS^._fZ2 := Z2;
END_SET
END_PROPERTY

END_FUNCTION_BLOCK

// ---- Shared/FB_SoComponent.TcPOU
(*
Abstract function block providing an :attr:`Output` property for single-output
controller toolbox components.

Concrete implementations must call this block cyclically and write their
result to ``_fOutput``.

.. note::
   Direct calls to this function block are not permitted (``no_explicit_call``).
   Extend it and call the derived block instead.
*)
{attribute 'no_explicit_call' := 'direct call for this function block is not allowed'}
FUNCTION_BLOCK ABSTRACT FB_SoComponent
IMPLEMENTS I_SoComponent
VAR
	_fOutput : LREAL;
END_VAR

(* Gets the output produced by the component.*)
PROPERTY Output : LREAL
GET
Output := THIS^._fOutput;
END_GET
END_PROPERTY

END_FUNCTION_BLOCK

// ---- Control/FB_ProportionalGain.TcPOU
(*
Applies a proportional gain to the input error signal.

The output is computed as:

.. math::

   y = K_p \cdot e

where :math:`K_p` is :attr:`Kp` and :math:`e` is the error signal set via :attr:`Input`.

.. note::
   The block is ``FINAL`` and must be instantiated, not extended.
   Use ``FB_init`` to set :attr:`fKp` at declaration time.
*)
{attribute 'no_assign'}
{attribute 'enable_dynamic_creation'}
{attribute 'no_explicit_call' := 'direct call for this function block is not allowed'}
FUNCTION_BLOCK FINAL FB_ProportionalGain EXTENDS FB_SisoComponent
IMPLEMENTS FsCommon.I_Runnable, I_Resettable
VAR
	_fKp : LREAL; // Proportional gain.
END_VAR

METHOD FB_init : BOOL
VAR_INPUT
	bInitRetains : BOOL; // if TRUE, the retain variables are initialized (warm start / cold start)
	bInCopyCode  : BOOL;  // if TRUE, the instance afterwards gets moved into the copy code (online change)
	fKp          : LREAL; // Proportional gain.
END_VAR
THIS^._fKp := fKp;
END_METHOD

(*
Gets or sets the proportional gain.

A higher value produces a stronger response to error but may cause overshoot.
A lower value produces a more gradual response. A value of 0 disables the
proportional term entirely.
*)
PROPERTY Kp : LREAL
GET
Kp := THIS^._fKp;
END_GET
SET
THIS^._fKp := Kp;
END_SET
END_PROPERTY

(* Sets the output to zero. Takes effect until the next :meth:`Run` call. *)
METHOD Reset
VAR_INPUT
END_VAR
THIS^._fOutput := 0;
END_METHOD

(*
Computes the proportional output for the current cycle.

.. note::
   Must be called once per cycle on a single PLC task.
*)
METHOD Run
VAR_INPUT
END_VAR
THIS^._fOutput := THIS^._fKp * THIS^._fInput;
END_METHOD

END_FUNCTION_BLOCK

// ---- Control/FB_TrackingIntegrator.TcPOU
(*
Integrates the input error signal with back-calculation anti-windup.

Extends :class:`FB_Integrator` by accepting an external comparator input,
typically the :attr:`~FB_Clamp.Residual` of an :class:`FB_Clamp` block, to
unwind the integrator gradually when the output is saturated. The residual is
scaled by ``1 / Tt`` and subtracted from the integrator input each cycle.

A typical wiring pattern:

.. code-block:: pascal

   fbI.Input           := fbP.Output; // Standard form. Use fError for parallel form.
   fbI.ComparatorInput := fbClamp.Residual;
   fbI.Run();
   fbClamp.Input := fbP.Output + fbI.Output + fbD.Output;
   fbClamp.Run();

.. note::
   Set :attr:`Maximum` before :attr:`Minimum` to ensure the clamp guard applies
   correctly.

   Use ``FB_init`` to set :attr:`tTn` and :attr:`tTt` at declaration time.
*)
{attribute 'no_assign'}
{attribute 'enable_dynamic_creation'}
{attribute 'no_explicit_call' := 'direct call for this function block is not allowed'}
FUNCTION_BLOCK FINAL FB_TrackingIntegrator EXTENDS FB_Integrator
VAR
	_fComparatorInput  : LREAL; // External residual signal for back-calculation anti-windup.
	_tTt 			   : LTIME; // Tracking time constant (Tt). Controls how quickly the integrator unwinds.
END_VAR

(*
Gets or sets the comparator input.

This is typically the :attr:`~FB_Clamp.Residual` of an :class:`FB_Clamp` block
placed after the PID summation, passed directly without negation. The block
subtracts the scaled residual from the integrator input internally to unwind
the integrator when the output is saturated.

A positive value indicates the unsaturated sum exceeded the clamp maximum.
A negative value indicates it fell below the clamp minimum.
*)
PROPERTY ComparatorInput : LREAL
GET
ComparatorInput := THIS^._fComparatorInput;
END_GET
SET
THIS^._fComparatorInput := ComparatorInput;
END_SET
END_PROPERTY

METHOD FB_init : BOOL
VAR_INPUT
	bInitRetains : BOOL;  // if TRUE, the retain variables are initialized (warm start / cold start)
	bInCopyCode  : BOOL;  // if TRUE, the instance afterwards gets moved into the copy code (online change)
	tTn          : LTIME; // Integral action time. LTIME#0 disables integration.
	tTt 		 : LTIME; // Tracking time constant (Tt). A typical starting value is SQRT(Tn * Td).
END_VAR
THIS^._tTt := tTt;
END_METHOD

(*
Advances the tracking integrator by one time step.

.. note::
   Must be called once per cycle on a single PLC task. If :attr:`Tn` is
   ``LTIME#0`` the output is set to zero. If :attr:`Tt` is ``LTIME#0``
   the back-calculation correction is disabled.
*)
METHOD Run
VAR_INST
	{attribute 'hide'}
	bInit       : BOOL := TRUE;
	{attribute 'hide'}
	fT          : LREAL;
	{attribute 'hide'}
	fbTaskCycle : FsCommon.FB_PlcTaskCycleChangeDetector(0);
END_VAR
VAR
	fKi         : LREAL;
	fTt         : LREAL;
	fWindupBack : LREAL;
END_VAR
IF bInit THEN
	fT := TO_LREAL(FsCommon.F_GetCurrentTaskCycleTime()) / TO_LREAL(LTIME#1S);
	RETURN(bInit := fT <= 0);
	fbTaskCycle.TaskIndex := FsCommon.F_GetCurrentTaskIndex();
END_IF

RETURN(NOT fbTaskCycle.HasChanged);

THIS^._fMaximum := MAX(THIS^._fMinimum, THIS^._fMaximum);
THIS^._fMinimum := MIN(THIS^._fMinimum, THIS^._fMaximum);

IF FsCommon.F_ResetOnTrue(THIS^._bSync) THEN
	THIS^._fOutput := LIMIT(THIS^._fMinimum, THIS^._fSync, THIS^._fMaximum);
END_IF

IF THIS^._tTn = LTIME#0S THEN
	THIS^._fOutput := 0;
	RETURN;
END_IF

fKi := 1.0 / (TO_LREAL(THIS^._tTn) / TO_LREAL(LTIME#1S));

IF THIS^._tTt > LTIME#0S THEN
	fTt         := TO_LREAL(THIS^._tTt) / TO_LREAL(LTIME#1S);
	fWindupBack := THIS^._fComparatorInput / fTt;
ELSE
	fWindupBack := 0;
END_IF

THIS^._fOutput := LIMIT(
	THIS^._fMinimum, 
	THIS^._fOutput + (fKi * THIS^._fInput - fWindupBack) * fT,
	THIS^._fMaximum
);
END_METHOD

(*
Gets or sets the tracking time constant (Tt).

Controls how quickly the integrator unwinds after saturation. A typical
starting value is ``SQRT(Tn * Td)``. Setting it to ``LTIME#0`` disables
the back-calculation correction entirely.
*)
PROPERTY Tt : LTIME
GET
Tt := THIS^._tTt;
END_GET
SET
THIS^._tTt := Tt;
END_SET
END_PROPERTY

END_FUNCTION_BLOCK

// ---- Filter/FB_FirstOrderIIRFilter.TcPOU
(*
Applies an exponential moving average (EMA) to the input signal.

On the first call the output is set to the current input. On subsequent calls:

.. math::

   y[k] = \alpha \cdot u[k] + (1 - \alpha) \cdot y[k-1]

where :math:`\alpha` is :attr:`Alpha`. A value of 0 passes the input through
unchanged. A value of 1 holds the output at the first input value.

.. note::
   The block is ``FINAL`` and must be instantiated, not extended.
   Use ``FB_init`` to set :attr:`fAlpha` at declaration time.
*)
{attribute 'no_assign'}
{attribute 'enable_dynamic_creation'}
{attribute 'no_explicit_call' := 'direct call for this function block is not allowed'}
FUNCTION_BLOCK FINAL FB_FirstOrderIIRFilter EXTENDS FB_SisoComponent
IMPLEMENTS FsCommon.I_Runnable, I_Resettable
VAR
	_fAlpha : LREAL; // Smoothing factor. Clamped to 0..1.
END_VAR

(*
Gets or sets the smoothing factor.

Controls the balance between the current input and the previous output.
A value closer to 0 produces a smoother, slower-responding output. A value
closer to 1 tracks the input more closely with less smoothing.
Values outside 0..1 are clamped.
*)
PROPERTY Alpha : LREAL
GET
Alpha := THIS^._fAlpha;
END_GET
SET
THIS^._fAlpha := LIMIT(0, Alpha, 1);
END_SET
END_PROPERTY

METHOD FB_init : BOOL
VAR_INPUT
	bInitRetains : BOOL; // if TRUE, the retain variables are initialized (warm start / cold start)
	bInCopyCode  : BOOL;  // if TRUE, the instance afterwards gets moved into the copy code (online change)
	fAlpha       : LREAL; // Smoothing factor. Clamped to 0..1.
END_VAR
THIS^._fAlpha := LIMIT(0, fAlpha, 1);
END_METHOD

(*
Sets the output to zero. 
On the next :meth:`Run` call the output will reinitialise to the current input.
*)
METHOD Reset
VAR_INPUT
END_VAR
THIS^._fOutput := 0;
END_METHOD

(*
Advances the filter by one time step.

On the first call the output is initialised to the current input to avoid
a transient caused by a zero initial state. Subsequent calls apply the
exponential moving average.
*)
METHOD Run
VAR_INST
	{attribute 'hide'}
	bInit : BOOL := TRUE;
END_VAR
IF FsCommon.F_ResetOnTrue(bInit) THEN
	THIS^._fOutput := THIS^._fInput;
	RETURN;
END_IF

THIS^._fOutput := THIS^._fAlpha * THIS^._fInput + (1.0 - THIS^._fAlpha) * THIS^._fOutput;
END_METHOD

END_FUNCTION_BLOCK

// ---- Project Information/F_GetCompany.TcPOU
// This function has been automatically generated from the project information.
{attribute 'signature_flag' := '1073741824'}
{attribute 'TcGenerated'}
{attribute 'no-analysis'}
FUNCTION F_GetCompany : WSTRING
VAR_INPUT
	
END_VAR

F_GetCompany := "FisoThemes";

END_FUNCTION

// ---- Project Information/F_GetTitle.TcPOU
// This function has been automatically generated from the project information.
{attribute 'signature_flag' := '1073741824'}
{attribute 'TcGenerated'}
{attribute 'no-analysis'}
FUNCTION F_GetTitle : WSTRING
VAR_INPUT
	
END_VAR

F_GetTitle := "FsControllerToolbox";

END_FUNCTION

// ---- Project Information/F_GetVersion.TcPOU
// This function has been automatically generated from the project information.
{attribute 'signature_flag' := '1073741824'}
{attribute 'TcGenerated'}
{attribute 'no-analysis'}
FUNCTION F_GetVersion : ST_LibVersion
VAR_INPUT
	
END_VAR

F_GetVersion.iMajor := 0;
F_GetVersion.iMinor := 4;
F_GetVersion.iBuild := 0;
F_GetVersion.iRevision := 0;
F_GetVersion.sVersion := '0.4.0';
F_GetVersion.nFlags := 0;

END_FUNCTION

// ---- Signals/FB_GaussianNoise.TcPOU
(*
Generates normally distributed (Gaussian) noise using the Box-Muller transform.

The output follows a normal distribution with the configured :attr:`Mean` and
:attr:`StdDev`. Values beyond ±3σ occur roughly 0.3% of the time. This models
real sensor noise more accurately than uniform white noise.

.. note::
   The block is ``FINAL`` and must be instantiated, not extended.
   Use ``FB_init`` to set :attr:`fMean` and :attr:`fStdDev` at declaration time.
*)
{attribute 'enable_dynamic_creation'}
{attribute 'no_explicit_call' := 'direct call for this function block is not allowed'}
FUNCTION_BLOCK FINAL FB_GaussianNoise EXTENDS FB_SoComponent
IMPLEMENTS FsCommon.I_Runnable
VAR
	_fMean   : LREAL; // Mean (centre) of the distribution.
	_fStdDev : LREAL; // Standard deviation. Controls the spread of the noise.
	_fbRng   : FsCommon.FB_RandomNumberGenerator(0); // Internal random number generator.
END_VAR

METHOD FB_init : BOOL
VAR_INPUT
	bInitRetains : BOOL; // if TRUE, the retain variables are initialized (warm start / cold start)
	bInCopyCode  : BOOL;  // if TRUE, the instance afterwards gets moved into the copy code (online change)
	fMean        : LREAL; // Mean of the distribution.
	fStdDev      : LREAL; // Standard deviation. A larger value produces more spread-out noise.
END_VAR
THIS^._fMean   := fMean;
THIS^._fStdDev := fStdDev;
END_METHOD

(*
Gets or sets the mean.

This is the centre of the distribution, the average value the noise oscillates
around. For pure noise centred on zero, set this to 0.
*)
PROPERTY Mean : LREAL
GET
Mean := THIS^._fMean;
END_GET
SET
THIS^._fMean := Mean;
END_SET
END_PROPERTY

(*
Generates the next Gaussian noise sample using the Box-Muller transform.

Two uniform random samples are drawn per cycle to produce one Gaussian sample.
If either sample is zero it is replaced with a small epsilon to avoid a
logarithm of zero.
*)
METHOD Run
VAR
	fU1       : LREAL;
	fU2       : LREAL;
	fEpsilon  : LREAL := 1.0E-10;
END_VAR
fU1 := ABS(THIS^._fbRng.NextReal());
fU2 := ABS(THIS^._fbRng.NextReal());

// Guard against log(0)
IF fU1 < fEpsilon THEN fU1 := fEpsilon; END_IF
IF fU2 < fEpsilon THEN fU2 := fEpsilon; END_IF

THIS^._fOutput := THIS^._fMean +
	THIS^._fStdDev * SQRT(-2.0 * LN(fU1)) * COS(2.0 * Tc2_System.PI * fU2);
END_METHOD

(*
Gets or sets the standard deviation (σ).

Controls the spread of the noise. Roughly 68% of samples fall within ±1σ of
the mean, 95% within ±2σ, and 99.7% within ±3σ. A larger value produces
more spread-out noise.
*)
PROPERTY StdDev : LREAL
GET
StdDev := THIS^._fStdDev;
END_GET
SET
THIS^._fStdDev := StdDev;
END_SET
END_PROPERTY

END_FUNCTION_BLOCK

// ---- Signals/FB_PeriodicSignal.TcPOU
(*
Abstract base block for periodic signal generators.

Provides :attr:`Period`, :attr:`Amplitude`, :attr:`Bias`, and :attr:`Phase`
as shared properties for all periodic signal generators. Derived blocks can
implement :meth:`Run` and :meth:`Reset` to produce their specific waveform.

.. note::
   Direct calls to this function block are not permitted (``no_explicit_call``).
   Extend it and call the derived block instead.
*)
{attribute 'enable_dynamic_creation'}
{attribute 'no_explicit_call' := 'direct call for this function block is not allowed'}
FUNCTION_BLOCK ABSTRACT FB_PeriodicSignal EXTENDS FB_SoComponent
IMPLEMENTS I_PeriodicSignal
VAR
	_tPeriod    : LTIME; // Duration of one full cycle. Must be greater than zero.
	_fAmplitude : LREAL; // Scales the raw wave. Output swings between Bias ± Amplitude.
	_fBias      : LREAL; // Shifts the output vertically.
	_fPhase     : LREAL; // Phase offset in radians. Shifts the wave horizontally.
END_VAR

(*
Gets or sets the amplitude. 

The output swings between ``Bias + Amplitude`` and ``Bias - Amplitude``.
*)
PROPERTY Amplitude : LREAL
GET
Amplitude := THIS^._fAmplitude;
END_GET
SET
THIS^._fAmplitude := Amplitude;
END_SET
END_PROPERTY

(*
Gets or sets the bias.

This is a fixed offset added to the output, shifting the wave up or down.
*)
PROPERTY Bias : LREAL
GET
Bias := THIS^._fBias;
END_GET
SET
THIS^._fBias := Bias;
END_SET
END_PROPERTY

(* 
Gets or sets the period. 

This is the time taken to complete one full cycle.
*)
PROPERTY Period : LTIME
GET
Period := THIS^._tPeriod;
END_GET
SET
THIS^._tPeriod := Period;
END_SET
END_PROPERTY

(*
Gets or sets the phase offset in radians.

This shifts the wave horizontally. Negative values shift in the opposite direction.
*)
PROPERTY Phase : LREAL
GET
Phase := THIS^._fPhase;
END_GET
SET
THIS^._fPhase := Phase;
END_SET
END_PROPERTY

END_FUNCTION_BLOCK

// ---- Signals/FB_PWM.TcPOU
(*
Generates a pulse-width modulated (PWM) signal.

The output switches between ``Amplitude`` and ``0`` at a fixed :attr:`Period`.
:attr:`DutyCycle` controls the proportion of the period the output is high,
as a value between -1 and 1.

For example, a duty cycle of 0.3 produces a high output for 30% of the period
and a low output for the remaining 70%. A duty cycle of -0.3 inverts this,
producing a low output for 30% and a high output for 70%.

A duty cycle of 0 keeps the output permanently low. A duty cycle of ±1 keeps
it permanently high.

:attr:`Phase` shifts the wave horizontally in radians. Negative values shift
in the opposite direction.
:attr:`Bias` shifts the output vertically.

.. note::
   The block is ``FINAL`` and must be instantiated, not extended.
   Use ``FB_init`` to set :attr:`tPeriod`, :attr:`fAmplitude`, :attr:`fBias`,
   and :attr:`fDutyCycle` at declaration time.
*)
{attribute 'enable_dynamic_creation'}
{attribute 'no_explicit_call' := 'direct call for this function block is not allowed'}
FUNCTION_BLOCK FINAL FB_PWM EXTENDS FB_PeriodicSignal
IMPLEMENTS FsCommon.I_Runnable, I_Resettable
VAR
	_fDutyCycle : LREAL; // Proportion of the period the output is high. Clamped to -1..1. Negative values invert the wave.
	_bIsHigh    : BOOL;  // TRUE when the output is in its high state, regardless of amplitude, bias, or phase.
	{attribute 'hide'}
	_tTime      : LTIME;
END_VAR

(*
Gets or sets the duty cycle as a value between -1 and 1.

This controls the proportion of the period the output is high. A value of 0.3
keeps the output high for 30% of the period. A negative value inverts the wave —
-0.3 keeps the output low for 30% and high for the remaining 70%. Values outside
-1..1 are clamped. Changes take effect immediately.
*)
PROPERTY DutyCycle : LREAL
GET
DutyCycle := THIS^._fDutyCycle;
END_GET
SET
THIS^._fDutyCycle := LIMIT(-1, DutyCycle, 1);
END_SET
END_PROPERTY

METHOD FB_init : BOOL
VAR_INPUT
	bInitRetains : BOOL; // if TRUE, the retain variables are initialized (warm start / cold start)
	bInCopyCode : BOOL;  // if TRUE, the instance afterwards gets moved into the copy code (online change)
	tPeriod      : LTIME; // Duration of one full cycle.
	fAmplitude   : LREAL; // High-state output level. Low state is always 0.
	fBias        : LREAL; // Shifts the output vertically.
	fDutyCycle   : LREAL; // Proportion of the period the output is high. Clamped to -1..1.
END_VAR
THIS^._tPeriod    := tPeriod;
THIS^._fAmplitude := fAmplitude;
THIS^._fBias      := fBias;
THIS^._fDutyCycle := LIMIT(-1.0, fDutyCycle, 1.0);
END_METHOD

(*
Gets whether the output is currently in its high state.

TRUE regardless of the values of :attr:`Amplitude`, :attr:`Bias`, or :attr:`Phase`.
*)
PROPERTY IsHigh  : BOOL
GET
IsHigh := THIS^._bIsHigh;
END_GET
END_PROPERTY

(* 
Restarts the wave from the beginning by resetting the accumulated time to zero.
The duty cycle, phase, amplitude, and bias are unaffected.
*)
METHOD Reset
VAR_INPUT
END_VAR
THIS^._tTime  := LTIME#0S;
THIS^._bIsHigh := FALSE;
END_METHOD

(*
Advances the PWM signal by one time step.

.. note::
   Must be called once per cycle on a single PLC task. If the measured cycle
   time is zero or :attr:`Period` is zero, the method returns early without
   updating the output.
*)
METHOD Run
VAR_INST
	{attribute 'hide'}
	bInit       : BOOL := TRUE;
	{attribute 'hide'}
	fT          : LREAL;
	{attribute 'hide'}
	fbTaskCycle : FsCommon.FB_PlcTaskCycleChangeDetector(0);
END_VAR
VAR
	fPeriod    : LREAL;
	fPhaseTime : LREAL;
	fCyclePos  : LREAL;
	fDuty      : LREAL;
END_VAR
IF bInit THEN
	fT := TO_LREAL(FsCommon.F_GetCurrentTaskCycleTime()) / TO_LREAL(LTIME#1S);
	RETURN(bInit := fT <= 0);
	fbTaskCycle.TaskIndex := FsCommon.F_GetCurrentTaskIndex();
END_IF

RETURN(THIS^._tPeriod <= LTIME#0S OR NOT fbTaskCycle.HasChanged);

THIS^._tTime := THIS^._tTime + TO_LTIME(LREAL_TO_ULINT(fT * 1.0E9));

fPeriod    := TO_LREAL(THIS^._tPeriod) / TO_LREAL(LTIME#1S);
fPhaseTime := TO_LREAL(THIS^._tTime) / TO_LREAL(LTIME#1S) + (THIS^._fPhase / (2.0 * Tc2_System.PI)) * fPeriod;
fCyclePos  := Tc2_Math.LMOD(fPhaseTime, fPeriod) / fPeriod;

THIS^._fDutyCycle := LIMIT(-1, THIS^._fDutyCycle, 1);

fDuty := ABS(THIS^._fDutyCycle);

IF THIS^._fDutyCycle >= 0.0 THEN
	THIS^._bIsHigh := fCyclePos < fDuty;
ELSE
	THIS^._bIsHigh := fCyclePos >= (1.0 - fDuty);
END_IF

IF THIS^._bIsHigh THEN
	THIS^._fOutput := THIS^._fAmplitude + THIS^._fBias;
ELSE
	THIS^._fOutput := THIS^._fBias;
END_IF
END_METHOD

END_FUNCTION_BLOCK

// ---- Signals/FB_Ramp.TcPOU
(*
Generates a ramp signal that rises or falls at a fixed rate indefinitely.

The output starts at :attr:`StartValue` and advances at :attr:`Rate` units per second.
A positive rate produces a rising ramp, a negative rate a falling ramp.
Changing :attr:`Rate` mid-run takes effect immediately.

Calling :meth:`Reset` returns the output to :attr:`StartValue`.

.. note::
   The block is ``FINAL`` and must be instantiated, not extended.
   Use ``FB_init`` to set :attr:`fStartValue` and :attr:`fRate` at declaration time.
*)
{attribute 'enable_dynamic_creation'}
{attribute 'no_explicit_call' := 'direct call for this function block is not allowed'}
FUNCTION_BLOCK FINAL FB_Ramp EXTENDS FB_SoComponent
IMPLEMENTS FsCommon.I_Runnable, I_Resettable
VAR
	_fStartValue : LREAL; // Initial output value. Restored on Reset.
	_fRate       : LREAL; // Rate of change in units per second. Negative values produce a falling ramp.
END_VAR

METHOD FB_init : BOOL
VAR_INPUT
	bInitRetains : BOOL;  // if TRUE, the retain variables are initialized (warm start / cold start)
	bInCopyCode  : BOOL;  // if TRUE, the instance afterwards gets moved into the copy code (online change)
	fStartValue  : LREAL; // Initial output value.
	fRate        : LREAL; // Rate of change in units per second. Negative values produce a falling ramp.
END_VAR
THIS^._fStartValue := fStartValue;
THIS^._fRate       := fRate;
END_METHOD

(*
Gets or sets the rate of change in units per second.

A positive value produces a rising ramp, a negative value a falling ramp.
Changes take effect immediately.
*)
PROPERTY Rate : LREAL
GET
Rate := THIS^._fRate;
END_GET
SET
THIS^._fRate := Rate;
END_SET
END_PROPERTY

(* Resets the output to the start value set in ``FB_init``. The rate is unaffected. *)
METHOD Reset
VAR_INPUT
END_VAR
THIS^._fOutput := THIS^._fStartValue;
END_METHOD

(*
Advances the ramp by one time step.

.. note::
   Must be called once per cycle on a single PLC task. If the measured cycle
   time is zero the method returns early without updating the output.
*)
METHOD Run
VAR_INST
	{attribute 'hide'}
	bInit : BOOL := TRUE;
	{attribute 'hide'}
	fT    : LREAL;
	{attribute 'hide'}
	fbTaskCycle : FsCommon.FB_PlcTaskCycleChangeDetector(0);
END_VAR
IF bInit THEN
	fT := TO_LREAL(FsCommon.F_GetCurrentTaskCycleTime()) / TO_LREAL(LTIME#1S);
	RETURN(bInit := fT <= 0);
	fbTaskCycle.TaskIndex := FsCommon.F_GetCurrentTaskIndex();
END_IF

RETURN(NOT fbTaskCycle.HasChanged);

THIS^._fOutput := THIS^._fOutput + THIS^._fRate * fT;
END_METHOD

(*
Gets or sets the start value.

This is the output value the ramp returns to after a :meth:`Reset`.
*)
PROPERTY StartValue  : LREAL
GET
StartValue := THIS^._fStartValue;
END_GET
SET
THIS^._fStartValue := StartValue;
END_SET
END_PROPERTY

END_FUNCTION_BLOCK

// ---- Signals/FB_RampProfile.TcPOU
(*
Generates a ramp signal that rises or falls toward a target value within a
configurable duration, then holds at the target.

The rate of change is derived automatically from :attr:`Target`, :attr:`StartValue`,
and :attr:`Duration`. Once the output is within one time step of the target it
snaps to the target and :attr:`IsComplete` becomes ``TRUE``. If :attr:`Target`
or :attr:`Duration` change mid-run the rate is recalculated immediately.

A duration of ``LTIME#0`` snaps the output to :attr:`Target` immediately.
If :attr:`Target` equals :attr:`StartValue`, :attr:`IsComplete` is ``TRUE``
from the first call.

Calling :meth:`Reset` returns the output to :attr:`StartValue` and clears
:attr:`IsComplete`.

.. note::
   The block is ``FINAL`` and must be instantiated, not extended.
   Use ``FB_init`` to set :attr:`fStartValue`, :attr:`fTarget`, and :attr:`tDuration`
   at declaration time.
*)
{attribute 'no_assign'}
{attribute 'enable_dynamic_creation'}
{attribute 'no_explicit_call' := 'direct call for this function block is not allowed'}
FUNCTION_BLOCK FINAL FB_RampProfile EXTENDS FB_SoComponent
IMPLEMENTS FsCommon.I_Runnable, I_Resettable
VAR
	_fStartValue : LREAL; // Initial output value. Restored on Reset.
	_fTarget     : LREAL; // Target value to ramp toward.
	_tDuration   : LTIME; // Time to reach the target from StartValue.
	_bIsComplete : BOOL;  // TRUE when the output has reached the target.
END_VAR

(*
Gets or sets the duration. 

This is the time taken to ramp from :attr:`StartValue` to :attr:`Target`.
``LTIME#0`` snaps the output to the target immediately. 
Changes take effect immediately.
*)
PROPERTY Duration : LTIME
GET
Duration := THIS^._tDuration;
END_GET
SET
THIS^._tDuration := Duration;
END_SET
END_PROPERTY

METHOD FB_init : BOOL
VAR_INPUT
	bInitRetains : BOOL; // if TRUE, the retain variables are initialized (warm start / cold start)
	bInCopyCode  : BOOL;  // if TRUE, the instance afterwards gets moved into the copy code (online change)
	fStartValue  : LREAL; // Initial output value.
	fTarget      : LREAL; // Target value to ramp toward.
	tDuration    : LTIME; // Time to reach the target from StartValue. LTIME#0 snaps immediately.
END_VAR
THIS^._fStartValue := fStartValue;
THIS^._fTarget     := fTarget;
THIS^._tDuration   := tDuration;
THIS^._fOutput     := fStartValue;
END_METHOD

(*
Gets whether the output has reached :attr:`Target`. 

Becomes ``TRUE`` when the output is within one time step of the target,
and ``FALSE`` again if :attr:`Target` changes and the output no longer matches.
*)
PROPERTY IsComplete : BOOL
GET
IsComplete := THIS^._bIsComplete;
END_GET
SET
THIS^._bIsComplete := IsComplete;
END_SET
END_PROPERTY

(* Returns the output to the start value set in ``FB_init`` and clears :attr:`IsComplete`. *)
METHOD Reset
VAR_INPUT
END_VAR
THIS^._fOutput     := THIS^._fStartValue;
THIS^._bIsComplete := FALSE;
END_METHOD

(*
Advances the ramp profile by one time step.

.. note::
   Must be called once per cycle on a single PLC task. If the measured cycle
   time is zero the method returns early without updating the output.
*)
METHOD Run
VAR_INST
	{attribute 'hide'}
	bInit       : BOOL := TRUE;
	{attribute 'hide'}
	fT          : LREAL;
	{attribute 'hide'}
	fbTaskCycle : FsCommon.FB_PlcTaskCycleChangeDetector(0);
END_VAR
VAR
	fRate      : LREAL;
	fStep      : LREAL;
	fRemaining : LREAL;
	fDuration  : LREAL;
END_VAR
IF bInit THEN
	fT := TO_LREAL(FsCommon.F_GetCurrentTaskCycleTime()) / TO_LREAL(LTIME#1S);
	RETURN(bInit := fT <= 0);
	fbTaskCycle.TaskIndex := FsCommon.F_GetCurrentTaskIndex();
END_IF

RETURN(NOT fbTaskCycle.HasChanged);

fRemaining := THIS^._fTarget - THIS^._fOutput;

IF THIS^._tDuration = LTIME#0S OR THIS^._fTarget = THIS^._fStartValue THEN
	THIS^._fOutput     := THIS^._fTarget;
	THIS^._bIsComplete := TRUE;
	RETURN;
END_IF

fDuration := TO_LREAL(THIS^._tDuration) / TO_LREAL(LTIME#1S);
fRate     := ABS(THIS^._fTarget - THIS^._fStartValue) / fDuration;
fStep     := fRate * fT;

IF ABS(fRemaining) <= fStep THEN
	THIS^._fOutput     := THIS^._fTarget;
	THIS^._bIsComplete := TRUE;
ELSE
	THIS^._fOutput     := THIS^._fOutput + fStep * SEL(fRemaining > 0, -1.0, 1.0);
	THIS^._bIsComplete := FALSE;
END_IF
END_METHOD

(*
Gets or sets the start value.

This is the output value the ramp returns to after a :meth:`Reset`.
*)
PROPERTY StartValue : LREAL
GET
StartValue := THIS^._fStartValue;
END_GET
SET
THIS^._fStartValue := StartValue;
END_SET
END_PROPERTY

(*
Gets or sets the target value. 

The output ramps toward this value within :attr:`Duration`. 
Changes take effect immediately, recalculating the rate.
*)
PROPERTY Target : LREAL
GET
Target := THIS^._fTarget;
END_GET
SET
THIS^._fTarget := Target;
END_SET
END_PROPERTY

END_FUNCTION_BLOCK

// ---- Signals/FB_SawtoothWave.TcPOU
(*
Generates a sawtooth wave signal.

The output rises linearly from ``-Amplitude`` to ``+Amplitude`` over one full
cycle then resets instantly, or falls from ``+Amplitude`` to ``-Amplitude``
depending on :attr:`Direction`. :attr:`Bias` shifts the output vertically.

:attr:`Phase` shifts the wave horizontally in radians. Negative values shift
in the opposite direction.

.. note::
   The block is ``FINAL`` and must be instantiated, not extended.
   Use ``FB_init`` to set :attr:`tPeriod`, :attr:`fAmplitude`, :attr:`fBias` and
   :attr:`fPhase` at declaration time.
*)
{attribute 'enable_dynamic_creation'}
{attribute 'no_explicit_call' := 'direct call for this function block is not allowed'}
FUNCTION_BLOCK FINAL FB_SawtoothWave EXTENDS FB_PeriodicSignal
IMPLEMENTS FsCommon.I_Runnable, I_Resettable
VAR
	_eDirection : E_RampDirection; // Direction of the sawtooth. Rising goes from -Amplitude to +Amplitude, Falling goes from +Amplitude to -Amplitude.
	{attribute 'hide'}
	_tTime      : LTIME;
END_VAR

(*
Gets or sets the direction of the sawtooth.

:attr:`~E_RampDirection.Rising` ramps from ``-Amplitude`` to ``+Amplitude``
before resetting. :attr:`~E_RampDirection.Falling` is the inverse.
Changes take effect immediately.
*)
PROPERTY Direction : E_RampDirection
GET
Direction := THIS^._eDirection;
END_GET
SET
THIS^._eDirection := Direction;
END_SET
END_PROPERTY

METHOD FB_init : BOOL
VAR_INPUT
	bInitRetains : BOOL; // if TRUE, the retain variables are initialized (warm start / cold start)
	bInCopyCode : BOOL;  // if TRUE, the instance afterwards gets moved into the copy code (online change)
	tPeriod      : LTIME; // Duration of one full cycle.
	fAmplitude   : LREAL; // Scales the wave. Output swings between Bias ± Amplitude.
	fBias        : LREAL; // Shifts the output vertically.
	fPhase       : LREAL; // Phase offset in radians. Shifts the wave horizontally.
END_VAR
THIS^._tPeriod    := tPeriod;
THIS^._fAmplitude := fAmplitude;
THIS^._fBias      := fBias;
THIS^._fPhase     := fPhase;
END_METHOD

(* Restarts the wave from the beginning by resetting the accumulated time to zero. The phase, amplitude, and bias are unaffected. *)
METHOD Reset
VAR_INPUT
END_VAR
THIS^._tTime := LTIME#0S;
END_METHOD

(*
Advances the sawtooth wave by one time step.

.. note::
   Must be called once per cycle on a single PLC task. If the measured cycle
   time is zero or :attr:`Period` is zero, the method returns early without
   updating the output.
*)
METHOD Run
VAR_INST
	{attribute 'hide'}
	bInit       : BOOL := TRUE;
	{attribute 'hide'}
	fT          : LREAL;
	{attribute 'hide'}
	fbTaskCycle : FsCommon.FB_PlcTaskCycleChangeDetector(0);
END_VAR
VAR
	fPeriod     : LREAL;
	fPhaseTime  : LREAL;
	fCyclePos   : LREAL;
END_VAR
IF bInit THEN
	fT := TO_LREAL(FsCommon.F_GetCurrentTaskCycleTime()) / TO_LREAL(LTIME#1S);
	RETURN(bInit := fT <= 0);
	fbTaskCycle.TaskIndex := FsCommon.F_GetCurrentTaskIndex();
END_IF

RETURN(THIS^._tPeriod <= LTIME#0S OR NOT fbTaskCycle.HasChanged);

THIS^._tTime := THIS^._tTime + TO_LTIME(LREAL_TO_ULINT(fT * 1.0E9));

fPeriod    := TO_LREAL(THIS^._tPeriod) / TO_LREAL(LTIME#1S);
fPhaseTime := TO_LREAL(THIS^._tTime) / TO_LREAL(LTIME#1S) + (THIS^._fPhase / (2.0 * Tc2_System.PI)) * fPeriod;
fCyclePos  := Tc2_Math.LMOD(fPhaseTime, fPeriod) / fPeriod;

CASE THIS^._eDirection OF
	E_RampDirection.Rising:
		THIS^._fOutput := THIS^._fAmplitude * (2.0 * fCyclePos - 1.0) + THIS^._fBias;
	E_RampDirection.Falling:
		THIS^._fOutput := THIS^._fAmplitude * (1.0 - 2.0 * fCyclePos) + THIS^._fBias;
END_CASE
END_METHOD

END_FUNCTION_BLOCK

// ---- Signals/FB_SineWave.TcPOU
(*
Generates a sine wave signal.

The output follows:

.. math::

   y(t) = A \sin\left(\frac{2\pi}{T} t + \phi\right) + B

where :math:`A` is :attr:`Amplitude`, :math:`T` is :attr:`Period` in seconds,
:math:`\phi` is :attr:`Phase` in radians, and :math:`B` is :attr:`Bias`.

.. note::
   The block is ``FINAL`` and must be instantiated, not extended.
   Use ``FB_init`` to set :attr:`tPeriod`, :attr:`fAmplitude`, :attr:`fBias`,
   and :attr:`fPhase` at declaration time.
*)
{attribute 'enable_dynamic_creation'}
{attribute 'no_explicit_call' := 'direct call for this function block is not allowed'}
FUNCTION_BLOCK FINAL FB_SineWave EXTENDS FB_PeriodicSignal
IMPLEMENTS FsCommon.I_Runnable, I_Resettable
VAR
	{attribute 'hide'}
	_tTime : LTIME;
END_VAR

METHOD FB_init : BOOL
VAR_INPUT
	bInitRetains : BOOL; // if TRUE, the retain variables are initialized (warm start / cold start)
	bInCopyCode : BOOL;  // if TRUE, the instance afterwards gets moved into the copy code (online change)
	tPeriod      : LTIME; // Duration of one full cycle.
	fAmplitude   : LREAL; // Scales the wave. Output swings between Bias ± Amplitude.
	fBias        : LREAL; // Shifts the output vertically.
	fPhase       : LREAL; // Phase offset in radians. Shifts the wave horizontally.
END_VAR
THIS^._tPeriod    := tPeriod;
THIS^._fAmplitude := fAmplitude;
THIS^._fBias      := fBias;
THIS^._fPhase     := fPhase;
END_METHOD

(* Restarts the wave from the beginning by resetting the accumulated time to zero. The phase, amplitude, and bias are unaffected. *)
METHOD Reset
VAR_INPUT
END_VAR
THIS^._tTime := LTIME#0S;
END_METHOD

(*
Advances the sine wave by one time step.

.. note::
   Must be called once per cycle on a single PLC task. If the measured cycle
   time is zero or :attr:`Period` is zero, the method returns early without
   updating the output.
*)
METHOD Run
VAR_INST
	{attribute 'hide'}
	bInit       : BOOL := TRUE;
	{attribute 'hide'}
	fT          : LREAL;
	{attribute 'hide'}
	fbTaskCycle : FsCommon.FB_PlcTaskCycleChangeDetector(0);
END_VAR
VAR
	fPeriod : LREAL;
END_VAR
IF bInit THEN
	fT := TO_LREAL(FsCommon.F_GetCurrentTaskCycleTime()) / TO_LREAL(LTIME#1S);
	RETURN(bInit := fT <= 0);
	fbTaskCycle.TaskIndex := FsCommon.F_GetCurrentTaskIndex();
END_IF

RETURN(THIS^._tPeriod <= LTIME#0S OR NOT fbTaskCycle.HasChanged);

THIS^._tTime := THIS^._tTime + TO_LTIME(LREAL_TO_ULINT(fT * 1.0E9));

fPeriod := TO_LREAL(THIS^._tPeriod) / TO_LREAL(LTIME#1S);

THIS^._fOutput := THIS^._fAmplitude 
	* SIN((2.0 * Tc2_System.PI / fPeriod) * (TO_LREAL(THIS^._tTime) / TO_LREAL(LTIME#1S)) + THIS^._fPhase) 
	+ THIS^._fBias;
END_METHOD

END_FUNCTION_BLOCK

// ---- Signals/FB_SquareWave.TcPOU
(*
Generates a square wave signal.

The raw wave alternates between ``+1`` and ``-1`` over one period. :attr:`Amplitude`
scales the wave and :attr:`Bias` shifts it vertically, giving an output that swings
between ``Bias + Amplitude`` and ``Bias - Amplitude``.

:attr:`Phase` shifts the wave horizontally in radians. A phase of π starts the
wave in its low half-cycle, a phase of -π has the same effect.

.. note::
   The block is ``FINAL`` and must be instantiated, not extended.
   Use ``FB_init`` to set :attr:`tPeriod`, :attr:`fAmplitude`, :attr:`fBias`,
   and :attr:`fPhase` at declaration time.
*)
{attribute 'enable_dynamic_creation'}
{attribute 'no_explicit_call' := 'direct call for this function block is not allowed'}
FUNCTION_BLOCK FINAL FB_SquareWave EXTENDS FB_PeriodicSignal
IMPLEMENTS FsCommon.I_Runnable, I_Resettable
VAR
	{attribute 'hide'}
	_tTime : LTIME; // Accumulated time.
END_VAR

METHOD FB_init : BOOL
VAR_INPUT
	bInitRetains : BOOL;  // if TRUE, the retain variables are initialized (warm start / cold start)
	bInCopyCode  : BOOL;  // if TRUE, the instance afterwards gets moved into the copy code (online change)
	tPeriod      : LTIME; // Duration of one full cycle.
	fAmplitude   : LREAL; // Scales the ±1 wave. Output swings between Bias ± Amplitude.
	fBias        : LREAL; // Shifts the output up or down by a fixed value.
	fPhase       : LREAL; // Phase offset in radians. Shifts the wave horizontally. Negative values shift in the opposite direction.
END_VAR
THIS^._tPeriod    := tPeriod;
THIS^._fAmplitude := fAmplitude;
THIS^._fBias      := fBias;
THIS^._fPhase     := fPhase;
END_METHOD

(* Restarts the wave from the beginning by resetting the accumulated time to zero. The phase, amplitude, and bias are unaffected. *)
METHOD Reset
VAR_INPUT
END_VAR
THIS^._tTime := LTIME#0S;
END_METHOD

(*
Advances the square wave by one time step.

.. note::
   Must be called once per cycle on a single PLC task. If the measured cycle
   time is zero or :attr:`Period` is zero, the method returns early without
   updating the output.
*)
METHOD Run
VAR_INST
	{attribute 'hide'}
	bInit 		 : BOOL := TRUE;
	{attribute 'hide'}
	tT           : LTIME;
	{attribute 'hide'}
	fbTaskCycle  :  FsCommon.FB_PlcTaskCycleChangeDetector(0);
END_VAR
VAR
	fCyclePhase  : LREAL;
	fPeriod		 : LREAL;
END_VAR
IF bInit THEN
	tT := FsCommon.F_GetCurrentTaskCycleTime();
	RETURN(bInit := tT = LTIME#0S);
	fbTaskCycle.TaskIndex := FsCommon.F_GetCurrentTaskIndex();
END_IF

RETURN(THIS^._tPeriod <= LTIME#0S OR NOT fbTaskCycle.HasChanged);

THIS^._tTime := THIS^._tTime + tT;

fPeriod := TO_LREAL(THIS^._tPeriod) / TO_LREAL(LTIME#1S);

fCyclePhase := Tc2_Math.LMOD(
	(TO_LREAL(THIS^._tTime) / TO_LREAL(LTIME#1S)) + ((THIS^._fPhase / (2.0 * Tc2_System.PI)) * fPeriod), 
	fPeriod
) / fPeriod;

IF fCyclePhase < 0.5 THEN
	THIS^._fOutput :=  THIS^._fAmplitude + THIS^._fBias;
ELSE
	THIS^._fOutput := -THIS^._fAmplitude + THIS^._fBias;
END_IF
END_METHOD

END_FUNCTION_BLOCK

// ---- Signals/FB_TriangleWave.TcPOU
(*
Generates a triangle wave signal.

The output rises linearly from ``-Amplitude`` to ``+Amplitude`` over the first
half-cycle, then falls back to ``-Amplitude`` over the second half. :attr:`Bias`
shifts the output vertically.

:attr:`Phase` shifts the wave horizontally in radians. A phase of π starts the
wave at its peak rather than its trough.

.. note::
   The block is ``FINAL`` and must be instantiated, not extended.
   Use ``FB_init`` to set :attr:`tPeriod`, :attr:`fAmplitude`, :attr:`fBias`,
   and :attr:`fPhase` at declaration time.
*)
{attribute 'enable_dynamic_creation'}
{attribute 'no_explicit_call' := 'direct call for this function block is not allowed'}
FUNCTION_BLOCK FINAL FB_TriangleWave EXTENDS FB_PeriodicSignal
IMPLEMENTS FsCommon.I_Runnable, I_Resettable
VAR
	{attribute 'hide'}
	_tTime : LTIME;
END_VAR

METHOD FB_init : BOOL
VAR_INPUT
	bInitRetains : BOOL; // if TRUE, the retain variables are initialized (warm start / cold start)
	bInCopyCode : BOOL;  // if TRUE, the instance afterwards gets moved into the copy code (online change)
	tPeriod      : LTIME; // Duration of one full cycle.
	fAmplitude   : LREAL; // Scales the wave. Output swings between Bias ± Amplitude.
	fBias        : LREAL; // Shifts the output vertically.
	fPhase       : LREAL; // Phase offset in radians. Shifts the wave horizontally.
END_VAR
THIS^._tPeriod    := tPeriod;
THIS^._fAmplitude := fAmplitude;
THIS^._fBias      := fBias;
THIS^._fPhase     := fPhase;
END_METHOD

(* Restarts the wave from the beginning by resetting the accumulated time to zero. The phase, amplitude, and bias are unaffected. *)
METHOD Reset
VAR_INPUT
END_VAR
THIS^._tTime := LTIME#0S;
END_METHOD

(*
Advances the triangle wave by one time step.

.. note::
   Must be called once per cycle on a single PLC task. If the measured cycle
   time is zero or :attr:`Period` is zero, the method returns early without
   updating the output.
*)
METHOD Run
VAR_INST
	{attribute 'hide'}
	bInit       : BOOL := TRUE;
	{attribute 'hide'}
	fT          : LREAL;
	{attribute 'hide'}
	fbTaskCycle : FsCommon.FB_PlcTaskCycleChangeDetector(0);
END_VAR
VAR
	fPeriod     : LREAL;
	fPhaseTime  : LREAL;
	fCyclePos   : LREAL;
END_VAR
IF bInit THEN
	fT := TO_LREAL(FsCommon.F_GetCurrentTaskCycleTime()) / TO_LREAL(LTIME#1S);
	RETURN(bInit := fT <= 0);
	fbTaskCycle.TaskIndex := FsCommon.F_GetCurrentTaskIndex();
END_IF

RETURN(THIS^._tPeriod <= LTIME#0S OR NOT fbTaskCycle.HasChanged);

THIS^._tTime := THIS^._tTime + TO_LTIME(LREAL_TO_ULINT(fT * 1.0E9));

fPeriod    := TO_LREAL(THIS^._tPeriod) / TO_LREAL(LTIME#1S);
fPhaseTime := TO_LREAL(THIS^._tTime) / TO_LREAL(LTIME#1S) + (THIS^._fPhase / (2.0 * Tc2_system.PI)) * fPeriod;
fCyclePos  := Tc2_Math.LMOD(fPhaseTime, fPeriod) / fPeriod;

IF fCyclePos < 0.5 THEN
	THIS^._fOutput := THIS^._fAmplitude * (4.0 * fCyclePos - 1.0) + THIS^._fBias;
ELSE
	THIS^._fOutput := THIS^._fAmplitude * (3.0 - 4.0 * fCyclePos) + THIS^._fBias;
END_IF
END_METHOD

END_FUNCTION_BLOCK

// ---- Signals/FB_WhiteNoise.TcPOU
(*
Generates uniformly distributed white noise.

The output is a random value in the range [-:attr:`Amplitude`, +:attr:`Amplitude`]
on every cycle. Useful for testing controller robustness against measurement noise
and disturbances.

.. note::
   The block is ``FINAL`` and must be instantiated, not extended.
   Use ``FB_init`` to set :attr:`Amplitude` at declaration time.
*)
{attribute 'enable_dynamic_creation'}
{attribute 'no_explicit_call' := 'direct call for this function block is not allowed'}
FUNCTION_BLOCK FINAL FB_WhiteNoise EXTENDS FB_SoComponent
IMPLEMENTS FsCommon.I_Runnable
VAR
	_fAmplitude : LREAL; // Maximum absolute output value.
	_fbRng      : FsCommon.FB_RandomNumberGenerator(0); // Internal random number generator.
END_VAR

(*
Gets or sets the amplitude.

The output is uniformly distributed in [-:attr:`Amplitude`, +:attr:`Amplitude`].
A value of 0 holds the output at zero.
*)
PROPERTY Amplitude : LREAL
GET
END_GET
SET
END_SET
END_PROPERTY

METHOD FB_init : BOOL
VAR_INPUT
	bInitRetains : BOOL;  // if TRUE, the retain variables are initialized (warm start / cold start)
	bInCopyCode  : BOOL;  // if TRUE, the instance afterwards gets moved into the copy code (online change)
	fAmplitude   : LREAL; // Maximum absolute output value.
END_VAR
THIS^._fAmplitude := fAmplitude;
END_METHOD

(* Generates the next white noise sample. *)
METHOD Run
VAR_INPUT
END_VAR
THIS^._fOutput := THIS^._fbRng.NextRangedReal(-THIS^._fAmplitude, THIS^._fAmplitude);
END_METHOD

END_FUNCTION_BLOCK

// ---- Simulation/FB_FirstOrderPlant.TcPOU
(*
Simulates a first-order linear plant using Euler's backward (implicit) discretisation.

The continuous-time transfer function is:

.. math::

   G(s) = \frac{K}{\tau s + 1}

which discretises to:

.. math::

   y[k] = \frac{\tau \cdot y[k-1] + K \cdot \Delta t \cdot u[k]}{\tau + \Delta t}

where :math:`K` is :attr:`Gain`, :math:`\tau` is :attr:`Tau` in seconds, and
:math:`\Delta t` is the task cycle time, measured automatically on the first call.

.. note::
   The block is ``FINAL`` and must be instantiated, not extended.
   Use ``FB_init`` to set :attr:`fGain` and :attr:`fTau` at declaration time.
*)
{attribute 'enable_dynamic_creation'}
{attribute 'no_explicit_call' := 'direct call for this function block is not allowed'}
FUNCTION_BLOCK FINAL FB_FirstOrderPlant EXTENDS FB_SisoComponent
IMPLEMENTS FsCommon.I_Runnable, I_Resettable
VAR
	_fGain 	: LREAL; // Steady-state gain (K). Ratio of output to input once the plant has fully settled.
	_tTau 	: LTIME; // Time constant (τ). Time for the step response to reach 63.2% of its final value.
END_VAR

METHOD FB_init : BOOL
VAR_INPUT
	bInitRetains 	: BOOL;  // if TRUE, the retain variables are initialized (warm start / cold start)
	bInCopyCode 	: BOOL;  // if TRUE, the instance afterwards gets moved into the copy code (online change)
	fGain 			: LREAL; // Steady-state gain (K). Ratio of output to input once the plant has fully settled.
	tTau 			: LTIME; // Time constant (τ). Time for the step response to reach 63.2% of its final value.
END_VAR
THIS^._fGain := fGain;
THIS^._tTau  := tTau;
END_METHOD

(*
Gets or sets the steady-state gain.

This is the factor by which a constant input is scaled to produce the output once
the plant has fully settled. For example, a gain of 2 with a constant input of 5
will eventually produce an output of 10.
*)
PROPERTY Gain : LREAL
GET
Gain := THIS^._fGain;
END_GET
SET
THIS^._fGain := Gain;
END_SET
END_PROPERTY

(* Sets the output to zero, returning the plant to its initial state. *)
METHOD Reset
VAR_INPUT
END_VAR
THIS^._fOutput := 0;
END_METHOD

(*
Advances the plant by one time step.

.. note::
   Must be called once per cycle on a single PLC task. This is because on the 
   first call, the cycle time is measured and stored for use in all subsequent calls. 
 
   If the measured cycle time is zero the method returns early without updating 
   the output, guarding against a divide-by-zero.
*)
METHOD Run
VAR_INST
	{attribute 'hide'}
	bInit 	: BOOL := TRUE;
	{attribute 'hide'}
	fDt			: LREAL;
	{attribute 'hide'}
	fbTaskCycle :  FsCommon.FB_PlcTaskCycleChangeDetector(0);
END_VAR
VAR
	fTau 		: LREAL;
END_VAR
IF bInit THEN
	fDt := TO_LREAL(FsCommon.F_GetCurrentTaskCycleTime()) / TO_LREAL(LTIME#1S);
	RETURN(bInit := fDt <= 0);
	fbTaskCycle.TaskIndex := FsCommon.F_GetCurrentTaskIndex();
END_IF

RETURN(NOT fbTaskCycle.HasChanged);

fTau := TO_LREAL(THIS^._tTau) / TO_LREAL(LTIME#1S);

THIS^._fOutput := 
	(fTau * THIS^._fOutput + THIS^._fGain * fDt * THIS^._fInput) 
	/ 
	(fTau + fDt);
END_METHOD

(* 
Gets or sets the time constant (τ).

This controls how quickly the plant responds to a change in input. 
A larger value means a slower response. It is the time taken for the 
output to reach 63.2% of its final value after a step change in input.
*)
PROPERTY Tau : LTIME
GET
Tau := THIS^._tTau;
END_GET
SET
THIS^._tTau := Tau;
END_SET
END_PROPERTY

END_FUNCTION_BLOCK

// ---- Simulation/FB_PadeDelay.TcPOU
(*
Approximates a transport delay (dead time) using a second-order Padé approximation.

The continuous-time transfer function is:

.. math::

   G(s) = \frac{1 - \frac{L}{2}s + \frac{L^2}{12}s^2}{1 + \frac{L}{2}s + \frac{L^2}{12}s^2}

where :math:`L` is :attr:`DelayTime` in seconds. The approximation is discretised
using the Tustin (bilinear) method with frequency pre-warping.

The output initially moves in the opposite direction to the input before settling
at the correct delayed value. This is a known characteristic of Padé approximations
and not a bug.

A delay of ``LTIME#0`` passes the input through unchanged.

.. note::
   The block is ``FINAL`` and must be instantiated, not extended.
   Use ``FB_init`` to set :attr:`tDelayTime` at declaration time.
*)
{attribute 'enable_dynamic_creation'}
{attribute 'no_explicit_call' := 'direct call for this function block is not allowed'}
FUNCTION_BLOCK FINAL FB_PadeDelay EXTENDS FB_SisoComponent
IMPLEMENTS FsCommon.I_Runnable, I_Resettable
VAR
	_tDelayTime : LTIME; // Approximate transport delay (L).
	{attribute 'hide'}
	_fY1        : LREAL; // y[k-1]
	{attribute 'hide'}
	_fY2        : LREAL; // y[k-2]
	{attribute 'hide'}
	_fU1        : LREAL; // u[k-1]
	{attribute 'hide'}
	_fU2        : LREAL; // u[k-2]
END_VAR

(*
Gets or sets the approximate transport delay.

This is the time between a change in the input and when that change appears
at the output. Longer values produce a more sluggish, harder-to-control process.
A value of ``LTIME#0`` passes the input through unchanged.

Note that the Padé approximation causes the output to initially move in the
opposite direction to the input. This effect is more pronounced for longer
delays relative to the cycle time.
*)
PROPERTY DelayTime : LTIME
GET
DelayTime := THIS^._tDelayTime;
END_GET
SET
THIS^._tDelayTime := DelayTime;
END_SET
END_PROPERTY

METHOD FB_init : BOOL
VAR_INPUT
	bInitRetains : BOOL;  // if TRUE, the retain variables are initialized (warm start / cold start)
	bInCopyCode  : BOOL;  // if TRUE, the instance afterwards gets moved into the copy code (online change)
	tDelayTime   : LTIME; // Approximate transport delay.
END_VAR
THIS^._tDelayTime := tDelayTime;
END_METHOD

(* Clears all internal state, returning the delay approximation to its initial conditions. *)
METHOD Reset
VAR_INPUT
END_VAR
THIS^._fY1     := 0;
THIS^._fY2     := 0;
THIS^._fU1     := 0;
THIS^._fU2     := 0;
THIS^._fOutput := 0;
END_METHOD

(*
Advances the Padé delay by one time step.

.. note::
   Must be called once per cycle on a single PLC task. If the measured cycle
   time is zero or :attr:`DelayTime` is ``LTIME#0`` the input passes through
   unchanged.
*)
METHOD Run
VAR_INST
	{attribute 'hide'}
	bInit       : BOOL := TRUE;
	{attribute 'hide'}
	fT          : LREAL;
	{attribute 'hide'}
	fbTaskCycle : FsCommon.FB_PlcTaskCycleChangeDetector(0);
END_VAR
VAR
	fL   : LREAL;
	fL2  : LREAL;
	fA0  : LREAL;
	fA1  : LREAL;
	fA2  : LREAL;
	fB0  : LREAL;
	fB1  : LREAL;
	fB2  : LREAL;
	fDen : LREAL;
END_VAR
IF bInit THEN
	fT := TO_LREAL(FsCommon.F_GetCurrentTaskCycleTime()) / TO_LREAL(LTIME#1S);
	RETURN(bInit := fT <= 0);
	fbTaskCycle.TaskIndex := FsCommon.F_GetCurrentTaskIndex();
END_IF

RETURN(NOT fbTaskCycle.HasChanged);

IF THIS^._tDelayTime = LTIME#0S THEN
	THIS^._fOutput := THIS^._fInput;
	RETURN;
END_IF

fL  := TO_LREAL(THIS^._tDelayTime) / TO_LREAL(LTIME#1S);
fL2 := fL * fL;

// Tustin discretisation of second-order Padé
// Continuous: (12 - 6Ls + L²s²) / (12 + 6Ls + L²s²)
fa0  := 12.0 * fT * fT + 6.0 * fL * fT * 2.0 + fL2 * 4.0;
fA1  := 24.0 * fT * fT - fL2 * 8.0;
fA2  := 12.0 * fT * fT - 6.0 * fL * fT * 2.0 + fL2 * 4.0;
fB0  := fA2;
fB1  := fA1;
fB2  := fA0;
fDen := fA0;

THIS^._fOutput :=
	(fB0 * THIS^._fInput + fB1 * THIS^._fU1 + fB2 * THIS^._fU2
	- fA1 * THIS^._fY1 - fA2 * THIS^._fY2) / fDen;

THIS^._fY2 := THIS^._fY1;
THIS^._fY1 := THIS^._fOutput;
THIS^._fU2 := THIS^._fU1;
THIS^._fU1 := THIS^._fInput;
END_METHOD

END_FUNCTION_BLOCK

// ---- Simulation/FB_SecondOrderPlant.TcPOU
(*
Simulates a second-order linear plant using the Tustin (bilinear) discretisation
with frequency pre-warping to preserve the natural frequency :attr:`Wn` exactly.

The continuous-time transfer function is:

.. math::

   G(s) = \frac{K \omega_n^2}{s^2 + 2 \zeta \omega_n s + \omega_n^2}

where :math:`K` is :attr:`Gain`, :math:`\omega_n` is :attr:`Wn`, and
:math:`\zeta` is :attr:`Zeta`.

.. note::
   The block is ``FINAL`` and must be instantiated, not extended.
   Use ``FB_init`` to set :attr:`fGain`, :attr:`fWn`, and :attr:`fZeta` at declaration time.
*)
{attribute 'enable_dynamic_creation'}
{attribute 'no_explicit_call' := 'direct call for this function block is not allowed'}
FUNCTION_BLOCK FINAL FB_SecondOrderPlant EXTENDS FB_SisoComponent
IMPLEMENTS FsCommon.I_Runnable, I_Resettable
VAR
	_fGain 	: LREAL; // Steady-state gain (K). Ratio of output to input once the plant has fully settled.
	_fWn 	: LREAL; // Natural frequency, rad/s), sets how fast the plant responds.
	_fZeta	: LREAL; // Damping ratio. Less than 1 gives overshoot, 1 is critically damped, greater than 1 is overdamped.
	{attribute 'hide'}
	_fY1    : LREAL; // y[k-1]
	{attribute 'hide'}
    _fY2    : LREAL; // y[k-2]
	{attribute 'hide'}
    _fU1    : LREAL; // u[k-1]
	{attribute 'hide'}
    _fU2    : LREAL; // u[k-2]
END_VAR

METHOD FB_init : BOOL
VAR_INPUT
	bInitRetains : BOOL;  // if TRUE, the retain variables are initialized (warm start / cold start)
	bInCopyCode  : BOOL;  // if TRUE, the instance afterwards gets moved into the copy code (online change)
	fGain 		 : LREAL; // Steady-state gain (K). Ratio of output to input once the plant has fully settled.
	fWn 		 : LREAL; // Natural frequency in rad/s. Controls how fast the plant responds.
	fZeta 		 : LREAL; // Damping ratio. Less than 1 gives overshoot, 1 is critically damped, greater than 1 is overdamped.
END_VAR
THIS^._fGain := fGain;
THIS^._fWn 	 := fWn;
THIS^._fZeta := fZeta;
END_METHOD

(*
Gets or sets the steady-state gain.

This is the factor by which a constant input is scaled to produce the output once
the plant has fully settled. For example, a gain of 2 with a constant input of 5
will eventually produce an output of 10.
*)
PROPERTY Gain : LREAL
GET
Gain := THIS^._fGain;
END_GET
SET
THIS^._fGain := Gain;
END_SET
END_PROPERTY

(* Sets the output and all internal state to zero, returning the plant to its initial conditions. *)
METHOD Reset
VAR_INPUT
END_VAR
THIS^._fOutput := 0;
THIS^._fY1     := 0;
THIS^._fY2     := 0;
THIS^._fU1     := 0;
THIS^._fU2     := 0;
END_METHOD

(*
Advances the plant by one time step.

.. note::
   Must be called once per cycle on a single PLC task. This is because on the 
   first call, the cycle time is measured and stored for use in all subsequent calls. 
 
   If the cycle time is zero or :attr:`Wn` is zero, the method returns early 
   without updating the output.
*)
METHOD Run
VAR_INST
	{attribute 'hide'}
	bInit 		 	: BOOL := TRUE;
	{attribute 'hide'}
	fT				 	: LREAL;
	{attribute 'hide'}
	fbTaskCycle 		:  FsCommon.FB_PlcTaskCycleChangeDetector(0);
END_VAR
VAR
	fWd, fWd2, fT2, fDen  : LREAL;
    fA1, fA2         : LREAL;
    fB0, fB1, fB2    : LREAL;
    fY               : LREAL;
END_VAR
IF bInit THEN
	fT := TO_LREAL(FsCommon.F_GetCurrentTaskCycleTime()) / TO_LREAL(LTIME#1S);
	RETURN(bInit := fT <= 0);
	fbTaskCycle.TaskIndex := FsCommon.F_GetCurrentTaskIndex();
	END_IF

RETURN(THIS^._fWn <= 0 OR NOT fbTaskCycle.HasChanged);

// Pre-warp natural frequency to preserve Wn exactly under Tustin
fWd  := (2.0 / fT) * TAN(THIS^._fWn * fT / 2.0);
fWd2 := fWd * fWd;
fT2  := fT * fT;
fDen := (4.0 / fT2) + 2.0 * THIS^._fZeta * fWd * (2.0 / fT) + fWd2;

fB0 := (THIS^._fGain * fWd2) / fDen;
fB1 := (2.0 * THIS^._fGain * fWd2) / fDen;
fB2 := fB0;

fA1 := ((-8.0 / fT2) + 2.0 * fWd2) / fDen;
fA2 := ((4.0 / fT2) - 2.0 * THIS^._fZeta * fWd * (2.0 / fT) + fWd2) / fDen;

fY := fB0 * THIS^._fInput + fB1 * THIS^._fU1 + fB2 * THIS^._fU2
       - fA1 * THIS^._fOutput - fA2 * THIS^._fY1;

THIS^._fY2      := THIS^._fY1;
THIS^._fY1      := THIS^._fOutput;
THIS^._fU2      := THIS^._fU1;
THIS^._fU1      := THIS^._fInput;
THIS^._fOutput 	:= fY;
END_METHOD

(*
Gets or sets the natural frequency in rad/s.

This controls the speed of the plant's response. 
A higher value means a faster response. To convert from Hz, multiply by 2π.
*)
PROPERTY Wn : LREAL
GET
Wn := THIS^._fWn;
END_GET
SET
THIS^._fWn := Wn;
END_SET
END_PROPERTY

(* 
Gets or sets the damping ratio.

This controls the shape of the response.
  - A value below 1 produces an oscillating response that overshoots before settling. 
  - A value of exactly 1 (critically damped) settles as fast as possible without any overshoot.
  - A value above 1 settles more slowly with no overshoot.
*)
PROPERTY Zeta : LREAL
GET
Zeta := THIS^._fZeta;
END_GET
SET
THIS^._fZeta := Zeta;
END_SET
END_PROPERTY

END_FUNCTION_BLOCK

// ---- Transform/FB_Bias.TcPOU
(*
Adds a fixed offset to the input signal.

A positive value shifts the output up; a negative value shifts it down.
*)
{attribute 'enable_dynamic_creation'}
{attribute 'no_explicit_call' := 'direct call for this function block is not allowed'}
FUNCTION_BLOCK FINAL FB_Bias EXTENDS FB_SisoComponent
IMPLEMENTS FsCommon.I_Runnable
VAR
	_fBias : LREAL; // Fixed offset added to the input.
END_VAR

(* Gets or sets the fixed offset added to the input. Negative values subtract. *)
PROPERTY Bias : LREAL
GET
Bias := THIS^._fBias;
END_GET
SET
THIS^._fBias := Bias;
END_SET
END_PROPERTY

METHOD FB_init : BOOL
VAR_INPUT
	bInitRetains : BOOL; // if TRUE, the retain variables are initialized (warm start / cold start)
	bInCopyCode  : BOOL;  // if TRUE, the instance afterwards gets moved into the copy code (online change)
	fBias        : LREAL; // Fixed offset added to the input.
END_VAR
THIS^._fBias := fBias;
END_METHOD

(* Adds :attr:`Bias` to the current input. *)
METHOD Run
VAR_INPUT
END_VAR
THIS^._fOutput := THIS^._fInput + THIS^._fBias;
END_METHOD

END_FUNCTION_BLOCK

// ---- Transform/FB_Gain.TcPOU
(*
Scales the input signal by a fixed gain.

A value greater than 1 amplifies the signal. A value between 0 and 1 attenuates
it. A negative value inverts and scales. A value of 0 holds the output at zero.
*)
{attribute 'enable_dynamic_creation'}
{attribute 'no_explicit_call' := 'direct call for this function block is not allowed'}
FUNCTION_BLOCK FINAL FB_Gain EXTENDS FB_SisoComponent
IMPLEMENTS FsCommon.I_Runnable
VAR
	_fGain : LREAL; // Factor the input is scaled by.
END_VAR

METHOD FB_init : BOOL
VAR_INPUT
	bInitRetains : BOOL; // if TRUE, the retain variables are initialized (warm start / cold start)
	bInCopyCode  : BOOL;  // if TRUE, the instance afterwards gets moved into the copy code (online change)
	fGain        : LREAL; // Factor the input is scaled by.
END_VAR
THIS^._fGain := fGain;
END_METHOD

(*
Gets or sets the scaling factor.

A value greater than 1 amplifies the signal. A value between 0 and 1
attenuates it. A value of -1 inverts the signal. A value of 0 holds
the output at zero.
*)
PROPERTY Gain : LREAL
GET
Gain := THIS^._fGain;
END_GET
SET
THIS^._fGain := Gain;
END_SET
END_PROPERTY

(* Scales the current input by :attr:`Gain`. *)
METHOD Run
VAR_INPUT
END_VAR
THIS^._fOutput := THIS^._fInput * THIS^._fGain;
END_METHOD

END_FUNCTION_BLOCK

// ---- Transform/FB_LinearScaler.TcPOU
(*
Maps the input signal from one range to another using linear interpolation.

The input range [:attr:`InputMin`, :attr:`InputMax`] is mapped to the output
range [:attr:`OutputMin`, :attr:`OutputMax`]. Values outside the input range
are extrapolated linearly.

If :attr:`InputMin` equals :attr:`InputMax` the output is set to :attr:`OutputMin`.

.. note::
   The block is ``FINAL`` and must be instantiated, not extended.
   Use ``FB_init`` to set :attr:`fInputMax`, :attr:`fInputMin`, :attr:`fOutputMin`,
   :attr:`fOutputMax` and :attr:`fOutputMin` at declaration time.
*)
{attribute 'enable_dynamic_creation'}
{attribute 'no_explicit_call' := 'direct call for this function block is not allowed'}
FUNCTION_BLOCK FINAL FB_LinearScaler EXTENDS FB_SisoComponent
IMPLEMENTS FsCommon.I_Runnable
VAR
	_fInputMax  : LREAL; // Upper bound of the input range.
	_fInputMin  : LREAL; // Lower bound of the input range.
	_fOutputMax : LREAL; // Upper bound of the output range.
	_fOutputMin : LREAL; // Lower bound of the output range.
END_VAR

METHOD FB_init : BOOL
VAR_INPUT
	bInitRetains : BOOL; // if TRUE, the retain variables are initialized (warm start / cold start)
	bInCopyCode  : BOOL;  // if TRUE, the instance afterwards gets moved into the copy code (online change)
	fInputMax    : LREAL; // Upper bound of the input range.
	fInputMin    : LREAL; // Lower bound of the input range.
	fOutputMax   : LREAL; // Upper bound of the output range.
	fOutputMin   : LREAL; // Lower bound of the output range.
END_VAR
THIS^._fInputMax  := fInputMax;
THIS^._fInputMin  := fInputMin;
THIS^._fOutputMax := fOutputMax;
THIS^._fOutputMin := fOutputMin;
END_METHOD

(* Gets or sets the upper bound of the input range. *)
PROPERTY InputMax : LREAL
GET
InputMax := THIS^._fInputMax;
END_GET
SET
THIS^._fInputMax := InputMax;
END_SET
END_PROPERTY

(* Gets or sets the lower bound of the input range. *)
PROPERTY InputMin : LREAL
GET
InputMin := THIS^._fInputMin;
END_GET
SET
THIS^._fInputMin := InputMin;
END_SET
END_PROPERTY

(* Gets or sets the upper bound of the output range. *)
PROPERTY OutputMax : LREAL
GET
OutputMax := THIS^._fOutputMax;
END_GET
SET
THIS^._fOutputMax := OutputMax;
END_SET
END_PROPERTY

(* Gets or sets the lower bound of the output range. *)
PROPERTY OutputMin : LREAL
GET
OutputMin := THIS^._fOutputMin;
END_GET
SET
THIS^._fOutputMin := OutputMin;
END_SET
END_PROPERTY

(* Applies the linear scaling to the current input. *)
METHOD Run
VAR_INPUT
END_VAR
IF THIS^._fInputMin = THIS^._fInputMax THEN
	THIS^._fOutput := THIS^._fOutputMin;
	RETURN;
END_IF

THIS^._fOutput := FsCommon.F_Lerp(
	THIS^._fOutputMin,
	THIS^._fOutputMax,
	(THIS^._fInput - THIS^._fInputMin) / (THIS^._fInputMax - THIS^._fInputMin));
END_METHOD

END_FUNCTION_BLOCK

// ---- Transform/FB_Quantizer.TcPOU
(*
Rounds the input signal to the nearest multiple of :attr:`StepSize`.

Useful for simulating ADC resolution, modelling actuators with discrete
positions, or testing controller behaviour under quantisation.

A :attr:`StepSize` of zero passes the input through unchanged.

.. note::
   The block is ``FINAL`` and must be instantiated, not extended.
   Use ``FB_init`` to set :attr:`fStepSize` at declaration time.
*)
{attribute 'enable_dynamic_creation'}
{attribute 'no_explicit_call' := 'direct call for this function block is not allowed'}
FUNCTION_BLOCK FINAL FB_Quantizer EXTENDS FB_SisoComponent
IMPLEMENTS FsCommon.I_Runnable
VAR
	_fStepSize : LREAL; // Quantisation step size. Zero passes the input through unchanged.
END_VAR

METHOD FB_init : BOOL
VAR_INPUT
	bInitRetains : BOOL; // if TRUE, the retain variables are initialized (warm start / cold start)
	bInCopyCode  : BOOL;  // if TRUE, the instance afterwards gets moved into the copy code (online change)
	fStepSize    : LREAL; // Quantisation step size. Zero passes the input through unchanged.
END_VAR
THIS^._fStepSize := fStepSize;
END_METHOD

(* Applies quantisation to the current input. *)
METHOD Run
VAR_INPUT
END_VAR
IF THIS^._fStepSize = 0 THEN
	THIS^._fOutput := THIS^._fInput;
	RETURN;
END_IF

THIS^._fOutput := FsCommon.F_TruncateNumber(
	THIS^._fInput / THIS^._fStepSize + 0.5
) * THIS^._fStepSize;
END_METHOD

(*
Gets or sets the quantisation step size.

The output is rounded to the nearest multiple of this value. For example,
a step size of 0.5 rounds the input to the nearest 0.5. A value of zero
passes the input through unchanged.
*)
PROPERTY StepSize : LREAL
GET
StepSize := THIS^._fStepSize;
END_GET
SET
THIS^._fStepSize := StepSize;
END_SET
END_PROPERTY

END_FUNCTION_BLOCK
